METHOD  M_STATE_DORMANT
VAR_INPUT
END_VAR
Busy    := FALSE;
Done    := FALSE;
Aborted := FALSE;
Error   := FALSE;
FeedBack.InterventionRequest :=FALSE;
strStatus :='FB_UpperFeedInConveyor: No Error';
uiExecutingStep :=0;
uiResettingStep	:=0;
NoFirstBoxDiameter:= SecondBox:=FALSE;
tonUpperConveyorTimeOut.IN := FALSE;
tonUpperConveyorDelay.IN :=FALSE;
tonUpperTimeOut.IN :=FALSE;
tonUpperTimeOutFive.IN :=FALSE;
tonWaitSecondBoxArriveTimeout.IN :=FALSE;
TON_CheckHaveBox.IN :=false;
tonFeedAirBlowtime.IN :=false;
bSecondBoxInCameraPos := FALSE;
_bForceUpperCV_Use := false;
_Abort := _Executed := _Error:= _ResetCompleted:=_AbortCompleted:=FALSE;
iMoveConveyor := 0;
uiFirstBoxDiameterStep  :=0;
uiSecondBoxAirBlowStep	:=0;
_UniqueErrorCode :='0';
// 重置暫停相關變數
_bPaused := FALSE;
_bPauseEdge := FALSE;
IF Execute THEN
	RobotService_CheckUPCVServicedone := FALSE;
	eSTATE:=STATE_EXECUTING;
END_IF
END_METHOD

METHOD  M_STATE_ERROR
VAR_INPUT
END_VAR
ERROR :=TRUE;
Busy :=FALSE;
UniqueErrorCode:=_UniqueErrorCode;
SUPER^.Status := strStatus;
_fbDiameterMovement.Execute := FALSE;


Motor.List.UpCV.M_MotorStop(); 
OutPut.bCamara_Blow :=FALSE;

IF NOT Execute THEN	
eSTATE:=STATE_RESETTING;
END_IF
END_METHOD

METHOD  M_STATE_EXECUTING
VAR_INPUT
END_VAR

VAR_INST
	
	
END_VAR
VAR
	END_I: INT;
	
END_VAR
// 如果暫停中，直接返回不執行
IF _bPaused THEN
	RETURN;
END_IF

Busy :=TRUE;

//Conveyor motor control
CASE iMoveConveyor OF
	1:
	Motor.list.UpCV.M_MoveForward();
	Cylinder.List.fbUpCV_CamaraPress4.M_Retract(); //Feedin working , open the end to allow box feedin
	//OutPut.bCamara_Blow :=TRUE;
	-1:
	Motor.list.UpCV.M_MoveBackward();
	Cylinder.List.fbUpCV_CamaraPress4.M_Retract(); //Feedin working , open the end to allow box feedin
ELSE		
	Motor.list.UpCV.M_MotorStop();
	Cylinder.List.fbUpCV_CamaraPress4.M_Extend();// End feedin , block the conveyor in case no one push boxes in working area
	//OutPut.bCamara_Blow :=FALSE;		change use airflow to take photo before
END_CASE



CASE uiExecutingStep OF
	
0 : // StandBy
	TON_RecordTimer.IN := TRUE;
	iMoveConveyor:=0;
	tonUpperConveyorTimeOut.IN:=FALSE;
	tonUpperConveyorDelay.IN :=FALSE;
	tonUpperConveyorDelay.PT:=T#200MS;
	IF Info.NrOfBox=1 THEN
		SecondBox:=FALSE;
	ELSIF Info.NrOfBox=2 THEN
		SecondBox:=TRUE;	
	ELSE
	_Error := TRUE;
	  strStatus := 'FB_UpperFeedInConveyor Step 0: Data not correct';
	END_IF
	uiExecutingStep :=10;

10: //Prepare cylinders
	IF Cylinder.List.fbUpCV_FeedInPress1.xError THEN
		Cylinder.List.fbUpCV_FeedInPress1.M_Reset();
	END_IF
	IF Cylinder.List.fbUpCV_FeedInPress2.xError THEN
		Cylinder.List.fbUpCV_FeedInPress1.M_Reset();
	END_IF
	IF Cylinder.List.fbUpCV_DiameterPress.xError THEN
		Cylinder.List.fbUpCV_DiameterPress.M_Reset();
	END_IF
	IF Cylinder.List.fbUpCV_CamaraPress1.xError THEN
		Cylinder.List.fbUpCV_CamaraPress1.M_Reset();
	END_IF
	IF Cylinder.List.fbUpCV_CamaraPress2.xError THEN
		Cylinder.List.fbUpCV_CamaraPress2.M_Reset();
	END_IF
	IF Cylinder.List.fbUpCV_CamaraPress4.xError THEN
		Cylinder.List.fbUpCV_CamaraPress4.M_Reset();
	END_IF
	IF Cylinder.List.fbUpCV_Block1.xError THEN
		Cylinder.List.fbUpCV_Block1.M_Reset();
	END_IF
	IF Cylinder.List.fbUpCV_Block2.xError THEN
		Cylinder.List.fbUpCV_Block2.M_Reset();
	END_IF
	IF Cylinder.List.fbUpCV_Block3.xError THEN
		Cylinder.List.fbUpCV_Block3.M_Reset();
	END_IF
	IF Motor.List.UpCV.xError THEN
		Motor.List.UpCV.M_Reset();
	END_IF
	
	uiExecutingStep :=20;
	
20: //Prepare cylinders
	tonUpperTimeOut.IN :=TRUE;
	Cylinder.List.fbUpCV_FeedInPress1.M_Retract();		(* Cylinder.List.fbUpCV_FeedInPress1.M_Retract();*)	
	Cylinder.List.fbUpCV_FeedInPress2.M_Retract();		(*Cylinder.List.fbUpCV_FeedInPress2.M_Retract();*)
	Cylinder.List.fbUpCV_DiameterPress.M_Retract();		(*Cylinder.List.fbUpCV_DiameterPress.M_Retract();*)
	Cylinder.List.fbUpCV_CamaraPress1.M_Retract();		(*Cylinder.List.fbUpCV_CamaraPress1.M_Retract();*)		
	//Cylinder.List.fbUpCV_CamaraPress2.M_Retract();	(*Cylinder.List.fbUpCV_CamaraPress2.M_Retract();*)
	Cylinder.List.fbUpCV_CamaraPress4.M_Retract();		(*Cylinder.List.fbUpCV_CamaraPress4.M_Retract();*)	
	Cylinder.List.fbUpCV_Block1.M_Retract();			(*Cylinder.List.fbUpCV_Block1.M_Retract();*)
	Cylinder.List.fbUpCV_Block2.M_Retract();			(*Cylinder.List.fbUpCV_Block2.M_Retract();*)
	Cylinder.List.fbUpCV_Block3.M_Retract();			(*Cylinder.List.fbUpCV_Block3.M_Retract();*)

	//edit by Min 20250326
	IF Cylinder.List.fbUpCV_FeedInPress1.InRearPosition AND		
		Cylinder.List.fbUpCV_FeedInPress2.InRearPosition AND
		Cylinder.List.fbUpCV_DiameterPress.InRearPosition AND
		Cylinder.List.fbUpCV_CamaraPress1.InRearPosition AND
		Cylinder.List.fbUpCV_CamaraPress4.InRearPosition AND
		Cylinder.List.fbUpCV_Block1.InRearPosition AND
		Cylinder.List.fbUpCV_Block2.InRearPosition AND
		Cylinder.List.fbUpCV_Block3.InRearPosition THEN
		
		tonUpperTimeOut.IN :=FALSE;
		uiExecutingStep :=100;	
	END_IF
	IF tonUpperTimeOut.Q THEN
		_Abort :=TRUE;
		strStatus :='FB_UpperFeedInConveyor Step 20: Prepare Cylinder clear command timeout';
	END_IF
	
100:// Check No Box 
	IF Input.bUpCV_Block1Detect_Sensor OR 
	  Input.bUpCV_Block2Detect_Sensor OR
	  Input.bUpCV_BoxArrived_Sensor OR
	  Input.bUpCV_Block3Detect_Sensor THEN
	 	 IF NOT AddingBox THEN
		 _bForceUpperCV_Use := TRUE;		//force UpperCV for Backward CV use
	 	 uiExecutingStep :=110; //Try reverse conveyor 
			ELSE 
			  _Abort := TRUE;
		 	 strStatus := 'FB_UpperFeedInConveyor Step 100: Conveyor not ready , please remove boxes in front';
		  END_IF
	 ELSE
 		uiExecutingStep :=200; 
	 END_IF
110:
		iMoveConveyor:= -1;
		Cylinder.List.fbUpCV_CamaraPress2.M_Retract();
		tonReverseConveyorDelay.IN :=TRUE;
		uiExecutingStep :=120;

120:
		//tonFeedAirBlowtime.IN :=TRUE;
		IF tonReverseConveyorDelay.Q THEN
			iMoveConveyor :=0;
			uiExecutingStep :=130; 
		END_IF
130:
		tonReverseConveyorDelay.IN :=FALSE;
		IF Input.bUpCV_Block1Detect_Sensor OR 
		  Input.bUpCV_Block2Detect_Sensor OR
		  Input.bUpCV_BoxArrived_Sensor OR
	 	 Input.bUpCV_Block3Detect_Sensor THEN
			  _Abort := TRUE;
		 	 strStatus := 'FB_UpperFeedInConveyor Step 130: Conveyor not ready , please remove boxes in front';
		 ELSE
			uiExecutingStep :=140; 	 
		 END_IF		
140:
   		IF Motor.list.UpCV.InStopped THEN
			uiExecutingStep :=200;
		END_IF
200: // motor start and camera block up 
	_bForceUpperCV_Use := FALSE;		//release UpperCV force use 
	tonUpperConveyorTimeOut.IN:=TRUE;
	iMoveConveyor:=1;
	Cylinder.List.fbUpCV_CamaraPress2.M_Retract();
	Cylinder.List.fbUpCV_Block3.M_Extend();
	IF Cylinder.List.fbUpCV_Block3.InFrontPosition AND
		Cylinder.List.fbUpCV_CamaraPress2.InRearPosition THEN
		tonUpperConveyorTimeOut.IN:=FALSE;
		uiExecutingStep :=300;
	END_IF
	IF tonUpperConveyorTimeOut.Q THEN
	  _Error := TRUE;
	  strStatus := 'FB_UpperFeedInConveyor Step 200: Cylinder.List.fbUpCV_Block3 timeout';
	END_IF
		  
	  
300://Dtect camera sensor and wait first box arrive in camera position
	TON_CheckHaveBox.IN :=TRUE;
	tonUpperConveyorDelay.IN:=Input.bUpCV_Block3Detect_Sensor; //Delay a moment to make sure box move till end of block 	
	IF tonUpperConveyorDelay.Q THEN
			TON_CheckHaveBox.IN :=FALSE;
			Cylinder.List.fbUpCV_CamaraPress1.M_Extend(); //Press box 
			tonUpperConveyorDelay.IN := FALSE;
			uiExecutingStep :=400;			
	END_IF
	IF TON_CheckHaveBox.Q THEN	//if behind not have box feedback box = 0
		uiExecutingStep := 2700;
	END_IF
	
400:// Check pressing job done for first box in camera position	
	tonUpperTimeOut.IN :=TRUE;
	IF Cylinder.List.fbUpCV_CamaraPress1.InFrontPosition THEN
		tonUpperTimeOut.IN := FALSE;
		Cylinder.List.fbUpCV_CamaraPress2.M_Extend();
		uiExecutingStep :=450;		
	END_IF
	IF tonUpperTimeOut.Q THEN
		_Abort := TRUE;
		strStatus := 'FB_UpperFeedInConveyor Step 400: Cylinder.List.fbUpCV_CamaraPress1.M_MoveForward timeout';
	END_IF

450:// send first box camera signal
	
	tonFeedAirBlowtime.IN :=TRUE;
	OutPut.bCamara_Blow :=TRUE;
	IF tonFeedAirBlowtime.Q THEN
		tonFeedAirBlowtime.IN:=FALSE;
		OutPut.bCamara_Blow :=FALSE;
		FeedBack.FirstBoxCamera :=TRUE;
		TON_RecordFirstTimer.IN :=TRUE;
		uiExecutingStep :=460;
	END_IF
	

460: // Wait first box camera done
	// todo : timeout
	tonUpperTimeOutFive.IN :=TRUE;		//T#5S
	IF Info.FirstBoxCameraDone THEN
		tonUpperTimeOutFive.IN :=FALSE;
		//FeedBack.FirstBoxCamera :=FALSE;
		uiExecutingStep :=500;
	END_IF	
	IF tonUpperTimeOutFive.Q THEN
		_Abort :=TRUE;
		strStatus := 'FB_UpperFeedInConveyor Step 460: C# FirstBoxCameraDone timeout';
	END_IF
	
500://Let first box move forward
	TSaveFirstTime 	:= TON_RecordFirstTimer.ET;
	TON_RecordFirstTimer .IN :=FALSE;
	Cylinder.List.fbUpCV_CamaraPress1.M_Retract(); // release press
	Cylinder.List.fbUpCV_Block3.M_Retract();//release blocker todo : add description
	uiExecutingStep :=550;
	
550://check cylinder inrearposition		edit by Min 20250326
	tonUpperTimeOut.IN :=TRUE;
	IF Cylinder.List.fbUpCV_CamaraPress1.InRearPosition AND		
		Cylinder.List.fbUpCV_Block3.InRearPosition THEN
		
		uiExecutingStep :=600;
	END_IF
	IF tonUpperTimeOut.Q THEN
		_Abort := TRUE;
		strStatus := 'FB_UpperFeedInConveyor Step 550: Cylinder.List.fbUpCV_CamaraPress1 or Cylinder.List.fbUpCV_Block3 InRearPosition timeout';
	END_IF
	
600://Check if diameter camera needed
	tonUpperTimeOut.IN :=FALSE;
	tonUpperTimeOutFive.IN :=TRUE;
	IF Info.FirstBoxCameraDiameterRequest THEN
		tonUpperTimeOutFive.IN :=FALSE;
		uiExecutingStep :=700;
		ELSE
			IF SecondBox THEN
				tonUpperTimeOutFive.IN :=FALSE;
				NoFirstBoxDiameter:=TRUE;
				uiExecutingStep :=610;//Only if box 1 no need to measure diameter
			ELSE
				tonUpperTimeOutFive.IN :=FALSE;
				uiExecutingStep :=2400;	
			END_IF
	END_IF
	IF tonUpperTimeOutFive.Q THEN
		_Abort := TRUE;
		strStatus :='FB_UpperFeedInConveyor Step 600: C# FirstBoxCameraDiameterRequest timeout';
	END_IF
	
610: //Check Box 1 leave read code camera position
	tonUpperTimeOut.IN :=TRUE;
	tonUpperConveyorDelay.IN := NOT Input.bUpCV_Block3Detect_Sensor;
	IF tonUpperConveyorDelay.Q THEN
		tonUpperConveyorDelay.IN :=FALSE;
		uiExecutingStep :=620;
	END_IF
	IF tonUpperTimeOut.Q  THEN
		_Abort :=TRUE;
		strStatus :='FB_UpperFeedInConveyor Step 610: Input.bUpCV_Block3Detect_Sensor first box leave timeout';
	END_IF
	
620: // Leave Box 2				//timeout and Check InRearPositonEdit by Min 20250326	
		tonUpperTimeOut.IN :=FALSE;	
		IF SecondBox THEN			
			Cylinder.List.fbUpCV_CamaraPress2.M_Retract(); //Release press box
			Cylinder.List.fbUpCV_Block3.M_Extend(); //release blocker
			IF Cylinder.List.fbUpCV_CamaraPress2.InRearPosition AND Cylinder.List.fbUpCV_Block3.InFrontPosition THEN
				uiExecutingStep :=1100;
			END_IF
		END_IF
		
700: //Rise diameter blocker
	tonUpperTimeOut.IN :=TRUE;
	Cylinder.List.fbUpCV_Block2.M_Extend();
	IF Cylinder.List.fbUpCV_Block2.InFrontPosition THEN
		tonUpperTimeOut.IN :=FALSE;
		uiExecutingStep :=800;
	END_IF
	IF tonUpperTimeOut.Q THEN
		_Abort :=TRUE;
		strStatus :='FB_UpperFeedInConveyor Step 700: Cylinder.List.fbUpCV_Block2 MoveForward timeout';
	END_IF
800: // wait first box ready on diameter position
	tonUpperTimeOut.IN :=TRUE;
	tonUpperConveyorDelay.IN:=Input.bUpCV_Block2Detect_Sensor;
	IF tonUpperConveyorDelay.Q THEN
		tonUpperTimeOut.IN :=FALSE;
		tonUpperConveyorDelay.IN:=FALSE;
		Cylinder.List.fbUpCV_DiameterPress.M_Extend();
		
		IF SecondBox THEN	
			tonUpperTimeOut.IN :=FALSE;		
			Cylinder.List.fbUpCV_CamaraPress2.M_Retract();
			Cylinder.List.fbUpCV_Block3.M_Extend();
		END_IF
		uiExecutingStep :=1000;
	END_IF
	IF tonUpperTimeOut.Q THEN
		_Abort :=TRUE;
		strStatus :='FB_UpperFeedInConveyor Step 800: Box not at Input.bUpCV_Block2Detect_Sensor ';
	END_IF
	
1000: // Wait diameter blocker ready
	tonUpperTimeOut.IN :=TRUE;
	IF 	Cylinder.List.fbUpCV_DiameterPress.InFrontPosition THEN
		tonUpperTimeOut.IN :=FALSE;
		uiExecutingStep :=1100;
	END_IF
	IF tonUpperTimeOut.Q THEN
		_Abort :=TRUE;
		strStatus :='FB_UpperFeedInConveyor Step 1000: Cylinder.List.fbUpCV_DiameterPress MoveForward timeout';
	END_IF

1100: // Pick needle to diameter camera

		
		CASE uiFirstBoxDiameterStep OF
			
		0:
			IF NOT NoFirstBoxDiameter THEN
	  			_fbDiameterMovement.Execute := TRUE;
				uiFirstBoxDiameterStep:=100;
			ELSE
				uiFirstBoxDiameterStep:=9000;	
	  		END_IF
		
		100:
			IF _fbDiameterMovement.Busy THEN
				uiFirstBoxDiameterStep:=200;
			END_IF	
			
		200:
			tonUpperTimeOutFive.IN :=TRUE;
			 IF _fbDiameterMovement.PickDone THEN
				  tonUpperTimeOutFive.IN :=FALSE;
				  FeedBack.FirstBoxCameraDiameter:=TRUE;		  
			  END_IF
			 IF Info.FirstBoxCameraDiameterDone THEN
				tonUpperTimeOutFive.IN:=FALSE;
				 FeedBack.FirstBoxCameraDiameter:=FALSE;
			 	_fbDiameterMovement.bContinue:=TRUE;
			 	uiFirstBoxDiameterStep:=300;
			  END_IF
			 IF tonUpperTimeOutFive.Q THEN
				 _Error :=TRUE;
				 strStatus :='FB_UpperFeedInConveyor Step 1100: box1 diameter timeout';
			 END_IF
		300:
			 IF _fbDiameterMovement.Done THEN
				  uiFirstBoxDiameterStep:=9000;		  
			  END_IF	  
		
		9000:
				_fbDiameterMovement.bContinue:=FALSE;
				_fbDiameterMovement.Execute:=FALSE;
				Cylinder.List.fbUpCV_DiameterPress.M_Retract();
				Cylinder.List.fbUpCV_Block2.M_Retract();
				// first box leave	  
				
				IF bSecondBoxInCameraPos AND 
					Cylinder.List.fbUpCV_DiameterPress.InRearPosition AND
					Cylinder.List.fbUpCV_Block2.InRearPosition THEN
					
					uiExecutingStep :=1200;
				END_IF
		END_CASE
						
		
	  		IF SecondBox THEN
				tonWaitSecondBoxArriveTimeout.IN :=TRUE;
	  			tonUpperConveyorDelay.IN := Input.bUpCV_Block3Detect_Sensor;
 				IF tonUpperConveyorDelay.Q THEN								
					tonUpperConveyorDelay.IN:=FALSE;
					tonWaitSecondBoxArriveTimeout.IN :=FALSE;
					Cylinder.List.fbUpCV_CamaraPress2.M_Extend();
					Cylinder.List.fbUpCV_CamaraPress1.M_Extend();
//					bSecondBoxInCameraPos :=TRUE;
				END_IF	
	 		 ELSE
				 bSecondBoxInCameraPos:=TRUE;
	 		 END_IF
			 
		CASE uiSecondBoxAirBlowStep OF
			 0:
			 	IF 	Cylinder.List.fbUpCV_CamaraPress1.InFrontPosition AND 
					Cylinder.List.fbUpCV_CamaraPress2.InFrontPosition THEN
						uiSecondBoxAirBlowStep :=10;
				END_IF
			10:
				OutPut.bCamara_Blow :=TRUE;		//take photo need airflow before
				tonFeedAirBlowtime.IN :=TRUE;
					IF tonFeedAirBlowtime.Q THEN		
						tonFeedAirBlowtime.IN :=FALSE;
						OutPut.bCamara_Blow :=FALSE;
						FeedBack.SecondBoxCamera:=TRUE;
						TON_RecordSecondTimer.IN :=TRUE;
						uiSecondBoxAirBlowStep :=20;
					END_IF
			20:
				IF Info.SecondBoxCameraDone THEN
					uiSecondBoxAirBlowStep :=30;
					TSaveSecondTime := TON_RecordSecondTimer.ET;
				END_IF
			30:	
					
					
					TON_RecordSecondTimer.IN :=FALSE;
					bSecondBoxInCameraPos:=TRUE;	
			
		END_CASE
		
//			IF Cylinder.List.fbUpCV_CamaraPress1.InFrontPosition AND 
//				Cylinder.List.fbUpCV_CamaraPress2.InFrontPosition THEN
//				OutPut.bCamara_Blow :=TRUE;		//take photo need airflow before
//				tonFeedAirBlowtime.IN :=TRUE;
//					IF tonFeedAirBlowtime.Q THEN		
//						tonFeedAirBlowtime.IN :=FALSE;
//						OutPut.bCamara_Blow :=FALSE;
//						FeedBack.SecondBoxCamera:=TRUE;	
//							IF Info.SecondBoxCameraDone THEN
//								bSecondBoxInCameraPos:=TRUE;	
//							END_IF	
//					END_IF
//			END_IF
	  
	  IF tonUpperConveyorTimeOut.Q THEN
			_Error :=TRUE;
			strStatus:='FB_UpperFeedInConveyor Step 1100: First box diameter timeout';		
		  
	  END_IF
		IF tonWaitSecondBoxArriveTimeout.Q THEN
			IF Input.bUpCV_ReLoadDetect_Sensor THEN
				_Error :=TRUE;
				strStatus:='FB_UpperFeedInConveyor Step 1100: Second box feedin to read code camera pos timeout';		
			ELSE
				tonUpperConveyorTimeOut.IN :=FALSE;
				SecondBox :=FALSE;
			END_IF	 
		END_IF

1200: 	// If first box leave diameter sensor , let second box go
		tonUpperTimeOut.IN :=TRUE;
		tonUpperConveyorDelay.PT:=T#600MS;		
		tonUpperConveyorDelay.IN := NOT Input.bUpCV_Block2Detect_Sensor;
		
		IF tonUpperConveyorDelay.Q THEN
			tonUpperConveyorDelay.IN :=FALSE;
			tonUpperTimeOut.IN :=FALSE;
			IF SecondBox AND INfo.SecondBoxCameraDiameterRequest THEN
				tonUpperTimeOut.IN :=FALSE;
				Cylinder.List.fbUpCV_Block2.M_Extend();
				Cylinder.List.fbUpCV_CamaraPress1.M_Retract();
				Cylinder.List.fbUpCV_Block3.M_Retract();
				uiExecutingStep :=1700;
			ELSE
				tonUpperTimeOut.IN :=FALSE;
				Cylinder.List.fbUpCV_CamaraPress1.M_Retract();
				Cylinder.List.fbUpCV_Block3.M_Retract();
				uiExecutingStep :=2400;	
			END_IF

		END_IF
		IF tonUpperTimeOut.Q THEN
			_Abort :=TRUE;
			strStatus :='FB_UpperFeedInConveyor Step 1200: First box still at Input.bUpCV_Block2Detect_Sensor';
		END_IF

1700: //Second box diameter request
		tonUpperTimeOut.IN :=TRUE;
		tonUpperConveyorDelay.IN :=Input.bUpCV_Block2Detect_Sensor;
		IF tonUpperConveyorDelay.Q THEN
			tonUpperTimeOut.IN :=FALSE;
			tonUpperConveyorDelay.IN :=FALSE;
			Cylinder.List.fbUpCV_DiameterPress.M_Extend();
			uiExecutingStep :=1800;
		END_IF
		IF tonUpperTimeOut.Q THEN
			_Abort :=TRUE;
			strStatus :='FB_UpperFeedInConveyor Step 1700: Input.bUpCV_Block2Detect_Sensor not have box';
		END_IF
1800: //wait second box in diameter position
		tonUpperTimeOut.IN :=TRUE;
		IF Cylinder.List.fbUpCV_DiameterPress.InFrontPosition THEN
			tonUpperTimeOut.IN :=FALSE;
			uiExecutingStep :=1900;
		END_IF
		IF tonUpperTimeOut.Q THEN
			_Abort :=TRUE;
			strStatus :='FB_UpperFeedInConveyor Step 1800: Cylinder.List.fbUpCV_DiameterPress MoveForward timeout';
			
		END_IF
		
1900:
		tonUpperTimeOutFive.IN :=TRUE;
		_fbDiameterMovement.Execute :=TRUE	;	
		IF _fbDiameterMovement.PickDone THEN
			tonUpperTimeOutFive.IN :=FALSE;
			FeedBack.SecondBoxCameraDiameter:=TRUE;
			uiExecutingStep :=2000;
		END_IF
		IF tonUpperTimeOutFive.Q THEN
			_Abort :=TRUE;
			strStatus :='FB_UpperFeedInConveyor Step 1900: C# DiameterMovement Pickdone timeout';
		END_IF
2000:	//check Second Box CamaraDone
		tonUpperTimeOutFive.IN :=TRUE;
		IF info.SecondBoxCameraDiameterDone THEN
			tonUpperTimeOutFive.IN :=FALSE;
			FeedBack.SecondBoxCameraDiameter:=FALSE;
			_fbDiameterMovement.bContinue:=TRUE;
			uiExecutingStep :=2100;
		END_IF
		IF tonUpperTimeOutFive.Q THEN
			_Abort :=TRUE;
			strStatus :='FB_UpperFeedInConveyor Step 2000: C# SecondBoxCameraDiameterDone timeout';
		END_IF		
2100:	
		tonUpperTimeOutFive.IN :=TRUE;
		IF _fbDiameterMovement.Done THEN
			tonUpperTimeOutFive.IN :=FALSE;
			_fbDiameterMovement.Execute:=FALSE;
			uiExecutingStep :=2150;
		END_IF
		IF tonUpperTimeOutFive.Q THEN
			_Abort :=TRUE;
			strStatus :='FB_UpperFeedInConveyor Step 2100: _fbDiameterMovement Done timeout';
		END_IF
2150:
		IF  Input.bUpCV_BoxArrived_Sensor  AND 
			NOT Input.bUpCV_Block1Detect_Sensor  THEN
			uiExecutingStep :=2200;
		END_IF
2200:	// release box 2 from diameter camera pos
		tonUpperTimeOut.IN :=TRUE;
		tonUpperConveyorDelay.PT:=T#100MS;
		tonUpperConveyorDelay.IN := NOT Input.bUpCV_Block1Detect_Sensor ;
		IF tonUpperConveyorDelay.Q THEN	
			tonUpperConveyorDelay.IN := FALSE;
			Cylinder.List.fbUpCV_Block1.M_Extend();
			Cylinder.List.fbUpCV_DiameterPress.M_Retract();		
			Cylinder.List.fbUpCV_Block2.M_Retract();
			uiExecutingStep :=2300;
		END_IF
		IF tonUpperTimeOut.Q THEN
			_Error :=TRUE;
			strStatus := 'FB_UpperFeedInConveyor Step 2200: There is a box on Input.bUpCV_Block1Detect_Sensor ';
		END_IF
		
		
2300:
		tonUpperTimeOut.IN :=TRUE;
		IF 	Cylinder.List.fbUpCV_DiameterPress.InRearPosition AND
			Cylinder.List.fbUpCV_Block1.InFrontPosition AND
			Cylinder.List.fbUpCV_Block2.InRearPosition THEN
			tonUpperTimeOut.IN :=FALSE;
			uiExecutingStep :=2500;
		END_IF	
		IF tonUpperTimeOut.Q THEN
			_Error :=TRUE;
			strStatus :='FB_UpperFeedInConveyor Step 2300: BlockBox1 MoveForward or BlockBox2 MoveBackward or DiameterMeasurementPressBox MoveBackward timeout';
		END_IF
2400:	//Check Box1 in FeedInBox1Detecting and Box2 leave BlockBox2Detecting
		
		tonUpperConveyorDelay.PT:=T#100MS;
		tonUpperConveyorDelay.IN := Input.bUpCV_BoxArrived_Sensor ;
		
		IF  tonUpperConveyorDelay.Q AND NOT Input.bUpCV_Block1Detect_Sensor  THEN
			tonUpperConveyorDelay.IN:=FALSE;
			Cylinder.List.fbUpCV_CamaraPress1.M_Retract();
			Cylinder.List.fbUpCV_Block3.M_Retract();
			Cylinder.List.fbUpCV_Block1.M_Extend();
			uiExecutingStep :=2500;
		END_IF
		
2500:	// Check Box1 in FeedInBox1Sensor and Box2 in BlockBox1Sensor
		tonUpperTimeOutFive.IN :=TRUE;
		tonUpperConveyorDelay.PT:=T#300MS;
		tonUpperConveyorDelay.IN := Input.bUpCV_BoxArrived_Sensor  AND 
		(Input.bUpCV_Block1Detect_Sensor  OR NOT SecondBox);
		
		IF tonUpperConveyorDelay.Q THEN
			tonUpperTimeOutFive.IN :=FALSE;
			tonUpperConveyorDelay.IN :=FALSE;
			Cylinder.List.fbUpCV_FeedInPress1.M_Extend();
			IF SecondBox THEN
				Cylinder.List.fbUpCV_FeedInPress2.M_Extend();
			END_IF
			uiExecutingStep :=2600;
		END_IF
		IF tonUpperTimeOutFive.Q THEN
			_Error :=TRUE;
			strStatus :='FB_UpperFeedInConveyor Step 2500: FeedInBox1Detecting not have a box';
		END_IF
2600:
		tonUpperConveyorDelay.PT:=T#500MS;
		tonUpperTimeOut.IN := TRUE;
		tonUpperConveyorDelay.IN :=  Cylinder.List.fbUpCV_FeedInPress1.InFrontPosition AND
		 (Cylinder.List.fbUpCV_FeedInPress2.InFrontPosition OR NOT SecondBox);		
//		IF tonUpperConveyorDelay.IN THEN
//			iMoveConveyor:=0;
//			//Motor.list.UpCV.M_StopMotor();
//		END_IF
		IF tonUpperConveyorDelay.Q THEN
			iMoveConveyor:=0;
			tonUpperTimeOut.IN :=FALSE;
			tonUpperConveyorDelay.IN :=FALSE;
			 Cylinder.List.fbUpCV_FeedInPress1.M_Retract();
			IF SecondBox THEN
				Cylinder.List.fbUpCV_FeedInPress2.M_Retract();
			END_IF
			uiExecutingStep :=2700;
		END_IF	
		IF tonUpperTimeOut.Q THEN
			_Error :=TRUE;
			strStatus :='FB_UpperFeedInConveyor Step 2600: Cylinder.List.fbUpCV_FeedInPress1 or Cylinder.List.fbUpCV_FeedInPress2 MoveForward timeout';
		END_IF
2700:
		tonUpperTimeOut.IN :=TRUE;
		IF TON_CheckHaveBox.IN THEN	// conveyor behind not have box feedback 0
			FeedBack.ActualNrOfBox:=0;
		ELSIF SecondBox THEN
			FeedBack.ActualNrOfBox:=2;
			ELSE
			FeedBack.ActualNrOfBox:=1;	
		END_IF
		//Cylinder.List.fbUpCV_Block1.M_Retract();
		//Cylinder.List.fbUpCV_CamaraPress2.M_Retract();
		IF NOT input.bUpCV_ReLoadDetect_Sensor  THEN
			FeedBack.InterventionRequest :=TRUE;
		END_IF
		IF// Cylinder.List.fbUpCV_Block1.InRearPosition AND
			 Cylinder.List.fbUpCV_FeedInPress1.InRearPosition AND
			Cylinder.List.fbUpCV_FeedInPress2.InRearPosition THEN
			//Cylinder.List.fbUpCV_CamaraPress2.InRearPosition THEN
			tonUpperTimeOut.IN :=FALSE;
			uiExecutingStep := 2800;
		END_IF	
		IF tonUpperTimeOut.Q THEN 
			_Error :=TRUE;
			strStatus :='FB_UpperFeedInConveyor Step 2700: FeedInPressBox1Cylinder or FeedInPressBox2Cylinder or ReadCodePressBox2Cylinder MoveBackward timeout';
		END_IF
		
2800:	//TO check the camera photo speed recoeding time
	TSaveTime 		:= TON_RecordTimer.ET;
	tRecordTimer[iArrayNumber] 			:=TSaveTime;
	tRecordFirstTimer[iArrayNumber] 	:=TSaveFirstTime;
	tRecordSecondTimer[iArrayNumber] 	:=TSaveSecondTime;
	uiExecutingStep := 2900;
2900:
	iArrayNumber := iArrayNumber+1;
	TON_RecordTimer.IN := FALSE;
	IF iArrayNumber >= 101 THEN
		bResetRecordInfo 	:=TRUE;
		iArrayNumber 		:=1;
	END_IF
	uiExecutingStep := 9999;
9999:
	bResetRecordInfo :=FALSE;
	TON_CheckHaveBox.IN :=FALSE;
	_Executed := TRUE;
				
END_CASE
	
	
IF NOT Execute THEN
	eState:=STATE_RESETTING;
END_IF
IF _Error THEN
	//FUN_UniqueErrorCodeGenerator(iErrorID := ErrorID,UinqueErrorCode=>_UniqueErrorCode);
	eState:=STATE_ERROR;
END_IF
IF _Abort OR Abort THEN
	//FUN_UniqueErrorCodeGenerator(iErrorID := ErrorID,UinqueErrorCode=>_UniqueErrorCode);
	eSTATE:=STATE_ABORTING;
END_IF
IF _Executed THEN
	eSTATE:=STATE_Done;
END_IF
END_METHOD

METHOD  M_STATE_RESETTING
VAR_INPUT
END_VAR
Error :=_Error;
Done :=_Executed;

tonUpperTimeOut.IN:=TRUE;
Motor.List.UpCV.M_MotorStop();

IF tonUpperTimeOut.Q OR NOT _Error THEN
	CASE uiResettingStep OF
		0: 
			IF _Error THEN
				Cylinder.List.fbUpCV_Block1.M_Retract();
			END_IF
			Cylinder.List.fbUpCV_FeedInPress1 .M_Retract();	
			Cylinder.List.fbUpCV_FeedInPress2.M_Retract();
			Cylinder.List.fbUpCV_DiameterPress.M_Retract();
			Cylinder.List.fbUpCV_CamaraPress1.M_Retract();	
			//UpperReadCodePressBox2Cylinder.M_Retract();	
			Cylinder.List.fbUpCV_Block2.M_Retract();	
			Cylinder.List.fbUpCV_Block3.M_Retract();	
			Cylinder.List.fbUpCV_CamaraPress4.M_Retract();
			OutPut.bCamara_Blow :=FALSE;
			_fbDiameterMovement.Execute := FALSE;
			_fbDiameterMovement.bContinue:=FALSE;
			FeedBack.InterventionRequest :=FALSE;
			FeedBack.FirstBoxCamera :=FALSE;
			FeedBack.FirstBoxCameraDiameter :=FALSE;
			FeedBack.SecondBoxCamera :=FALSE;
			FeedBack.SecondBoxCameraDiameter :=FALSE;

		
			uiResettingStep:=9999;
		
		9999:
			_ResetCompleted:=TRUE;
	END_CASE
END_IF
IF _ResetCompleted THEN
	eSTATE:=STATE_DORMANT;
END_IF
END_METHOD

END_FUNCTION_BLOCK

// ---- Library/20_MachineUnits/21_StorageArea/Service/FB_AddBoxes_v2.TcPOU
FUNCTION_BLOCK FB_AddBoxes_v2 EXTENDS FB_ObjectBase_V2
VAR_INPUT
//	UpperBoxRefillDetection		:REFERENCE TO FB_Sensor;
//	RackPusherCylinder			:REFERENCE TO FB_Cylinder;
//	RackMotor					:REFERENCE TO FB_RackMotor_V2;
//	bUpperLayerFeedInConveyor	:REFERENCE TO FB_Motor;
	Cylinder 	: REFERENCE TO UNI_CylinderList;
	Motor	 	: REFERENCE TO UNI_MotorList;
	Input 	 	: REFERENCE TO ST_InputTable;
	OutPut	 	: REFERENCE TO ST_OutputTable;
	CurrentData      : ST_SetupPara;

	ERackState	:E_RackState;
	bClearInterventionRequest : BOOL;
	_bForceUpperCV_Use		:BOOL;
END_VAR
VAR_OUTPUT
	InterventionRequest	 : BOOL;
	FeedingBoxes		:BOOL;
END_VAR
VAR
	RackMotorStationTable   : ARRAY[0..9] OF st_StationPositions;
	uiMaxRackStation :INT :=10;
//	eState :E_MethodStatus_Basic;
//	uiExecutingStep : UDINT; // This var is used to been controll STATE_EXECUTING process.
//	uiResettingStep : UDINT;
//	uiAbortingStep : UDINT;
//	_Executed :BOOL; // Executing process completed.
//	_Error : BOOL; // FB has an error.
//	_ResetCompleted : BOOL; // FB resetting completed.
//	_AbortCompleted : BOOL; // FB aborting completed.	

	tonAddBoxTimeOut	:TON;
	tonDetectSensor		:TON;
	tonConveyorTimeOut	:TON;
	tonFeedInUseAddBoxesDelay :TON;
	strStatus	:STRING;
//	_Abort		:BOOL;
	CurrStation : UINT;
	bInterventionRequest	 : BOOL;
	trigClearInterventionRequest : R_TRIG;
	_bClearInterventionRequestLast :BOOL;
	ftrigRackStateLeaveFeedBox		:F_Trig;
	_UniqueErrorCode : STRING;
	_RetryCompleted	 : BOOL; // FB Aboted STATE use

	// ===== Pause / Resume framework =====
	_bPaused					: BOOL;
	_bPauseEdge					: BOOL;

	// 計時器活動狀態保存
	bWasActive_tonAddBoxTimeOut			: BOOL;
	bWasActive_tonDetectSensor			: BOOL;
	bWasActive_tonConveyorTimeOut		: BOOL;
	bWasActive_tonFeedInUseAddBoxesDelay : BOOL;

	// 計時器剩餘時間保存
	tRemaining_tonAddBoxTimeOut			: TIME;
	tRemaining_tonDetectSensor			: TIME;
	tRemaining_tonConveyorTimeOut		: TIME;
	tRemaining_tonFeedInUseAddBoxesDelay : TIME;

	// 恢復後使用調整 PT 旗標 (Q 觸發或被外部關掉就清除)
	bUseAdjustedPT_tonAddBoxTimeOut		: BOOL;
	bUseAdjustedPT_tonDetectSensor		: BOOL;
	bUseAdjustedPT_tonConveyorTimeOut	: BOOL;
	bUseAdjustedPT_tonFeedInUseAddBoxesDelay : BOOL;

	// 馬達/輸出狀態保存
	bSaved_MoveConveyor			: BOOL;

	// 從 EXECUTING.VAR_INST 提到 FB-level (A01_PauseControl 需 access)
	bMoveConveyor				: BOOL;
END_VAR

A00_BasicUnits();
A01_PauseControl();

// 暫停時不執行狀態機
IF NOT _bPaused THEN
	SUPER^.A10_StateControl();
END_IF

ACTION A00_BasicUnits:
// 計時器 PT 設定 - 恢復後使用剩餘時間,完成後切回原 PT
IF bUseAdjustedPT_tonAddBoxTimeOut THEN
	tonAddBoxTimeOut(PT := tRemaining_tonAddBoxTimeOut);
	IF tonAddBoxTimeOut.Q OR NOT tonAddBoxTimeOut.IN THEN
		bUseAdjustedPT_tonAddBoxTimeOut := FALSE;
	END_IF
ELSE
	tonAddBoxTimeOut(PT:=T#120S);
END_IF

IF bUseAdjustedPT_tonDetectSensor THEN
	tonDetectSensor(PT := tRemaining_tonDetectSensor);
	IF tonDetectSensor.Q OR NOT tonDetectSensor.IN THEN
		bUseAdjustedPT_tonDetectSensor := FALSE;
	END_IF
ELSE
	tonDetectSensor(PT:=T#1S);
END_IF

IF bUseAdjustedPT_tonConveyorTimeOut THEN
	tonConveyorTimeOut(PT := tRemaining_tonConveyorTimeOut);
	IF tonConveyorTimeOut.Q OR NOT tonConveyorTimeOut.IN THEN
		bUseAdjustedPT_tonConveyorTimeOut := FALSE;
	END_IF
ELSE
	tonConveyorTimeOut(PT:=T#5S);
END_IF

IF bUseAdjustedPT_tonFeedInUseAddBoxesDelay THEN
	tonFeedInUseAddBoxesDelay(PT := tRemaining_tonFeedInUseAddBoxesDelay);
	IF tonFeedInUseAddBoxesDelay.Q OR NOT tonFeedInUseAddBoxesDelay.IN THEN
		bUseAdjustedPT_tonFeedInUseAddBoxesDelay := FALSE;
	END_IF
ELSE
	tonFeedInUseAddBoxesDelay(PT:=T#1S);
END_IF

ErrorID := 2700;

InterventionRequest:=bInterventionRequest;
ftrigRackStateLeaveFeedBox(CLK := (eRackState = E_RackState.FeedBox));
IF ftrigRackStateLeaveFeedBox.Q THEN
	bInterventionRequest:=FALSE;
END_IF

FeedingBoxes := eRackState=E_RackState.FeedBox;
END_ACTION

ACTION A01_PauseControl:
// A01_PauseControl - 暫停控制邏輯
// 依 PauseResume_Implementation_Guide.md 標準框架實作
// 控制對象: tonAddBoxTimeOut/tonDetectSensor/tonConveyorTimeOut/tonFeedInUseAddBoxesDelay 4 個計時器
//          Motor.List.UpCV (DC 馬達, 透過 bMoveConveyor 控制)
//          arAxisCtrl_gb[AxisNo.RackMotor] (伺服軸)

Paused := _bPaused;

// 只在執行狀態處理暫停
IF eState <> STATE_EXECUTING THEN
	_bPaused := FALSE;
	_bPauseEdge := FALSE;
	RETURN;
END_IF

// ===== 進入暫停 (上升邊緣) =====
IF Pause AND NOT _bPauseEdge THEN
	_bPauseEdge := TRUE;

	IF NOT _bPaused THEN
		_bPaused := TRUE;

		// 保存計時器活動狀態和剩餘時間
		bWasActive_tonAddBoxTimeOut := tonAddBoxTimeOut.IN;
		tRemaining_tonAddBoxTimeOut := T#120S - tonAddBoxTimeOut.ET;

		bWasActive_tonDetectSensor := tonDetectSensor.IN;
		tRemaining_tonDetectSensor := T#1S - tonDetectSensor.ET;

		bWasActive_tonConveyorTimeOut := tonConveyorTimeOut.IN;
		tRemaining_tonConveyorTimeOut := T#5S - tonConveyorTimeOut.ET;

		bWasActive_tonFeedInUseAddBoxesDelay := tonFeedInUseAddBoxesDelay.IN;
		tRemaining_tonFeedInUseAddBoxesDelay := T#1S - tonFeedInUseAddBoxesDelay.ET;

		// 停止所有計時器 (避免暫停期間 Timeout)
		tonAddBoxTimeOut.IN := FALSE;
		tonDetectSensor.IN := FALSE;
		tonConveyorTimeOut.IN := FALSE;
		tonFeedInUseAddBoxesDelay.IN := FALSE;

		// 保存上層輸送帶狀態
		bSaved_MoveConveyor := bMoveConveyor;

		// 停止上層輸送帶 (DC 馬達)
		Motor.List.UpCV.M_MotorStop();

		// 注意:RackMotor 不主動 halt
		// (1) 本 codebase 軸 API 沒有 Admin.Stop,要 halt 必須切 _OpMode.en := ModeAH 但 resume 後要重 issue 太複雜
		// (2) 暫停期間 SUPER^.A10_StateControl 不執行,軸完成 in-flight 移動後 state machine 不會推進
		// (3) Resume 時 step 210/610 直接看到 CmdDone 立即過 step,行為等價
	END_IF
END_IF

// ===== 離開暫停 (下降邊緣) - 必須等 Start 按鈕觸發 =====
IF NOT Pause AND _bPauseEdge AND GVL_ADS.OpPannel_Status.StartBtnStatus THEN
	_bPauseEdge := FALSE;

	IF _bPaused THEN
		_bPaused := FALSE;

		// 恢復上層輸送帶: 透過 bMoveConveyor 在 EXECUTING preamble 自動 M_MoveForward
		bMoveConveyor := bSaved_MoveConveyor;

		// 軸:暫停時沒主動 halt,resume 不需要 restore (對應上方 pause 注意事項)

		// 恢復計時器 (使用剩餘時間,A00 完成後切回原 PT)
		IF bWasActive_tonAddBoxTimeOut THEN
			bUseAdjustedPT_tonAddBoxTimeOut := TRUE;
			tonAddBoxTimeOut.IN := TRUE;
		END_IF

		IF bWasActive_tonDetectSensor THEN
			bUseAdjustedPT_tonDetectSensor := TRUE;
			tonDetectSensor.IN := TRUE;
		END_IF

		IF bWasActive_tonConveyorTimeOut THEN
			bUseAdjustedPT_tonConveyorTimeOut := TRUE;
			tonConveyorTimeOut.IN := TRUE;
		END_IF

		IF bWasActive_tonFeedInUseAddBoxesDelay THEN
			bUseAdjustedPT_tonFeedInUseAddBoxesDelay := TRUE;
			tonFeedInUseAddBoxesDelay.IN := TRUE;
		END_IF
	END_IF
END_IF

// 邊緣重置
IF NOT Pause THEN
	_bPauseEdge := FALSE;
END_IF
END_ACTION

METHOD PRIVATE M_CheckCommand : BOOL
VAR_INPUT
END_VAR
M_CheckCommand	:= true;
END_METHOD

METHOD PRIVATE M_GetCurrentStation : BOOL
VAR
	i : UINT;
	SetPos	 :LREAL;
END_VAR

VAR_OUTPUT
	uiCurrentStation	:UINT;
END_VAR
//SetPos := THIS^.fbMotor.NcToPlc.SetPos;
SetPos := arAxisCtrl_gb[AxisNo.RackMotor].Admin.Axis.NcToPlc.SetPos;
M_RefreshStationPos();
//IF  THIS^.fbMotor.Status.Homed THEN
IF arAxisCtrl_gb[AxisNo.RackMotor].Admin.Axis.Status.Homed THEN
	FOR i:=0 TO 9 BY 1 DO 
		IF SetPos> RackMotorStationTable[i].Position-5 AND SetPos< RackMotorStationTable[i].Position+5 THEN // Range should be confirm
			uiCurrentStation :=i;
			M_GetCurrentStation :=TRUE;
			RETURN;
		END_IF
	END_FOR
	
	uiCurrentStation:=99;
	M_GetCurrentStation :=FALSE;
ELSE
	M_GetCurrentStation :=FALSE;
	uiCurrentStation:=99;
END_IF
END_METHOD

METHOD PRIVATE M_MoveToStation : BOOL
VAR_INPUT
	uiStation : UINT;
END_VAR
VAR
	bDone	:BOOL;
	uiTargetPosition	:LREAL ;
END_VAR
M_RefreshStationPos();
IF uiStation>=0 AND uiStation <10 THEN
	uiTargetPosition :=RackMotorStationTable[uiStation].Position;
	
	arAxisCtrl_gb[AxisNo.RackMotor].PosMode.Acc := CurrentData.Axes.RackMotor.HalfAuto.Acceleration;
	arAxisCtrl_gb[AxisNo.RackMotor].PosMode.Dec := CurrentData.Axes.RackMotor.HalfAuto.Deceleration;
	arAxisCtrl_gb[AxisNo.RackMotor].PosMode.Jerk := CurrentData.Axes.RackMotor.HalfAuto.Jerk;
	arAxisCtrl_gb[AxisNo.RackMotor].PosMode.Velocity := CurrentData.Axes.RackMotor.HalfAuto.Velocity;
	arAxisCtrl_gb[AxisNo.RackMotor].PosMode.Position := uiTargetPosition;
	
//	THIS^.fbMotor.MoveAbs(lrPosition	:=uiTargetPosition,
//						lrVelocity 		:=GVL.MotorCore[AxisNo.RackMotor].VCC,
//						lrAcceleration	:=GVL.MotorCore[AxisNo.RackMotor].ACC,
//						lrDeceleration	:=GVL.MotorCore[AxisNo.RackMotor].DCC,
//						lrJerk			:=GVL.MotorCore[AxisNo.RackMotor].Jerk,
//						BufferMode		:=MC_BufferMode.MC_Aborting);
	//THIS^.fbMotor.GetCmdDoneStatus(bMotionCmdDone=>bDone);
ELSE
	M_MoveToStation :=FALSE;
	RETURN;
END_IF
END_METHOD

METHOD PRIVATE M_RefreshStationPos : BOOL
VAR_INPUT
END_VAR
VAR
	i: UINT;
	position : ST_PositionTable;
END_VAR
FOR i := 0 TO 9 DO
	position :=FUN_GetPositionTableData(PositionName:='W',Index:=i,Clip:=0);
RackMotorStationTable[i].Position:= position.X_Pos;
END_FOR
	M_RefreshStationPos :=TRUE;

// todo : update position of each stations
//FOR i:=1 TO 200 BY 1 DO
//	FOR iIndex:=0 TO 9 BY 1 DO
//		IF 		
//			DAS_CoreSys.MachineControl.CurrentData.PositionTable[i].Index= iIndex AND
//			DAS_CoreSys.MachineControl.CurrentData.PositionTable[i].Zone ='W' THEN
//			RackMotorStationTable[iIndex].Position := DAS_CoreSys.MachineControl.CurrentData.PositionTable[i].X_Pos;

//			StationsPosition[iIndex]:=RackMotorStationTable[i].Position;
//		ELSE
//			M_RefreshStationPos :=FALSE;
//		END_IF
//	END_FOR
//END_FOR
END_METHOD

METHOD  M_STATE_ABORTED
VAR_INPUT
END_VAR
Error :=TRUE;
Busy :=FALSE;
Done := FALSE;
Status :=strStatus;
UniqueErrorCode:=_UniqueErrorCode;
uiAbortingStep := 0;
_AbortCompleted := FALSE;


CASE uiExecutingStep OF
	0, 10:
			// init 階段 abort -> 從頭重跑
			_RetryCompleted := TRUE;
			uiExecutingStep := 0;
			strStatus := 'FB_AddBoxes_v2 init step: retrying from 0';

	100:
			_RetryCompleted := TRUE;
			uiExecutingStep := 100;
			strStatus := 'FB_AddBoxes_v2 Step 100: no error , retrying';

	200, 210:
			// 軸移動階段 abort -> 退到 200 重新發送移動指令
			_RetryCompleted := TRUE;
			uiExecutingStep := 200;
			strStatus := 'FB_AddBoxes_v2 Step 200/210: no error , retrying motion';

	300:
			_RetryCompleted := TRUE;
			uiExecutingStep := 300;
			strStatus := 'FB_AddBoxes_v2 Step 300: no error , retrying';

	400, 500:
			// sensor 檢查階段 abort -> 退到 400 重新檢查
			_RetryCompleted := TRUE;
			uiExecutingStep := 400;
			strStatus := 'FB_AddBoxes_v2 Step 400/500: no error , retrying refill check';

	600, 610:
			// 歸零移動階段 abort -> 退到 600 重新發送
			_RetryCompleted := TRUE;
			uiExecutingStep := 600;
			strStatus := 'FB_AddBoxes_v2 Step 600/610: no error , retrying home move';

	1000, 1100:
			// 收尾階段 abort -> 從 1000 完成停輸送帶
			_RetryCompleted := TRUE;
			uiExecutingStep := 1000;
			strStatus := 'FB_AddBoxes_v2 Step 1000/1100: no error , finishing';
ELSE
			// 未涵蓋的 step -> 不允許續作,只能放開 Execute 走 RESETTING 重跑
			_RetryCompleted := FALSE;
			strStatus := 'FB_AddBoxes_v2 unexpected step at aborted';
END_CASE

IF NOT Execute THEN
	eState := STATE_RESETTING;
END_IF

IF Execute AND Reset AND _RetryCompleted THEN
	_Abort := Error := _Error := FALSE;
	eState:=STATE_EXECUTING;
END_IF
END_METHOD

METHOD  M_STATE_ABORTING
VAR_INPUT
END_VAR
CASE uiAbortingStep of
	 0:		// 清空參數
			tonAddBoxTimeOut.IN			 := FALSE;
			tonDetectSensor.IN			 := FALSE;
			tonConveyorTimeOut.IN		 := FALSE;
			tonFeedInUseAddBoxesDelay.IN := FALSE;
			_RetryCompleted := FALSE;
			Motor.List.UpCV.M_MotorStop();
			
			uiAbortingStep := 100;
			
	100:	// 確認軸、氣缸是否有報錯
			IF  NOT arAxisCtrl_gb[AxisNo.RackMotor].Admin.Axis.Status.Error AND 
				NOT Cylinder.List.fbStackPush.xError THEN
				uiAbortingStep := 200;	
			ELSIF arAxisCtrl_gb[AxisNo.RackMotor].Admin.Axis.Status.Error THEN
				arAxisCtrl_gb[AxisNo.RackMotor].Admin.ClearError := TRUE;
			ELSIF Cylinder.List.fbStackPush.xError THEN
				Cylinder.List.fbStackPush.M_Reset();
			END_IF
			IF arAxisCtrl_gb[AxisNo.RackMotor].Admin.ClearError THEN 
				arAxisCtrl_gb[AxisNo.RackMotor].Admin.ClearError := FALSE;
			END_IF
			
	200:	// 推盒氣缸往後，料架軸
			Cylinder.List.fbStackPush.M_Retract();
			arAxisCtrl_gb[AxisNo.RackMotor].Admin._OpMode.en := E_AXIS_MODE.ModeAH;
			uiAbortingStep:=9999;
		
	9999:	
			_AbortCompleted:=TRUE;
END_CASE

IF	 _AbortCompleted THEN
	eSTATE:=STATE_ABORTED;
END_IF
END_METHOD

METHOD  M_STATE_DONE
VAR_INPUT
END_VAR
Busy := FALSE;
Done := TRUE;
IF NOT Execute THEN
	eState := STATE_RESETTING;
END_IF
END_METHOD

METHOD  M_STATE_DORMANT
VAR_INPUT
END_VAR
VAR
END_VAR
Busy    := FALSE;
Done    := FALSE;
Aborted := FALSE;
Error   := FALSE;
strStatus  := 'No error';
uiExecutingStep := 0;
uiResettingStep := 0;
uiAbortingStep:=0;
_ResetCompleted := FALSE;
_RetryCompleted := FALSE;
_AbortCompleted := FALSE;
_Abort := _Executed := _Error:= _ResetCompleted:=_AbortCompleted:=FALSE;
tonAddBoxTimeOut.IN :=FALSE;
tonDetectSensor.IN:=FALSE;
tonFeedInUseAddBoxesDelay.IN :=FALSE;
_UniqueErrorCode :='0';

// 重置暫停相關變數
_bPaused := FALSE;
_bPauseEdge := FALSE;

IF Execute  THEN
	IF eRackState = E_RackState.FeedBox THEN
		eState:= STATE_ERROR;
		strStatus :='FB_AddBoxes_v2: Rack occupied by user Push FeedButton';
		
	ELSIF  Input.bUpCV_ReLoadDetect_Sensor THEN
		_Executed :=TRUE;
		eState	:= STATE_Done;
	ELSE
		eState := STATE_EXECUTING;
	END_IF	
END_IF
END_METHOD

METHOD  M_STATE_ERROR
VAR_INPUT
END_VAR
Error := TRUE;
Busy :=FALSE;
Status :=strStatus;
UniqueErrorCode:=_UniqueErrorCode;

IF NOT Execute THEN
	eSTATE :=STATE_RESETTING;
END_IF

// 對稱 ABORTED 的 retry: 維持 Execute + 按 Reset 從 step 0 重跑
// 目前唯一 ERROR 觸發點 (step 0 wrong command) 由此處重試
IF Execute AND Reset THEN
	_Error := FALSE;
	Error := FALSE;
	uiExecutingStep := 0;
	eSTATE := STATE_EXECUTING;
END_IF
END_METHOD

METHOD  M_STATE_EXECUTING
VAR_INPUT
END_VAR
VAR_INST
	uiTargetStation	: UINT;
END_VAR
VAR
	bMotionDone : BOOL;
	
END_VAR
// 暫停中直接返回
IF _bPaused THEN
	RETURN;
END_IF

Busy := TRUE;
IF NOT _bForceUpperCV_Use THEN
	IF bMoveConveyor THEN
		Motor.List.UpCV.M_MoveForward();
//	ELSE
//		Motor.List.UpCV.M_MotorStop();
	END_IF
END_IF
CASE uiExecutingStep OF			
	
	0:	//check command
		tonAddBoxTimeOut.IN:=FALSE;
		tonFeedInUseAddBoxesDelay.IN :=TRUE;
		
		IF M_CheckCommand() THEN
			IF tonFeedInUseAddBoxesDelay.Q THEN
				tonFeedInUseAddBoxesDelay.IN :=FALSE;
				uiExecutingStep	:= 10 ;
			END_IF
		ELSE
			strStatus := 'FB_AddBoxes_v2 Step 0: Wrong command, check the command setting';
			_Error := TRUE;
		END_IF
	10:
		IF 	NOT	Motor.List.UpCV.InBackWard THEN
			uiExecutingStep	:= 100 ;
		END_IF
		//todo : Add timeout
		
 	100:	//release cylinder, check rackmotor currentStation
		tonAddBoxTimeOut.IN:=TRUE;
		tonDetectSensor.IN:=FALSE;
		Cylinder.List.fbStackPush.M_Retract();
		M_GetCurrentStation(uiCurrentStation =>CurrStation);
		
		IF	Cylinder.List.fbStackPush.InRearPosition THEN
			 CASE CurrStation OF
				0 ,99 :
					uiTargetStation:=1;				
				1,2,3,4,5,6,7,8,9 :
					uiTargetStation :=CurrStation;	
				ELSE // Error
					strStatus := 'FB_AddBoxes_v2 Step 100: Station get Error';
                    _Abort := TRUE;
			 END_CASE
			 
			 IF NOT _Abort THEN
                tonAddBoxTimeOut.IN := FALSE;
                uiExecutingStep := 200;
             END_IF
		END_IF
		
		IF tonAddBoxTimeOut.Q THEN
			strStatus := 'FB_AddBoxes_v2 Step 100: RackPusher move back timeout';
            _Abort := TRUE;
		END_IF
		
	200:	//check rackmotor station 
		tonDetectSensor.IN :=FALSE;
		IF uiTargetStation<10 THEN
			M_MoveToStation(uiTargetStation);
			uiExecutingStep := 210;	
		ELSE
			uiExecutingStep := 500;	
		END_IF
		
	
	210:
		tonAddBoxTimeOut.IN:=TRUE;
		bMotionDone:= arAxisStatus_gb[AxisNo.RackMotor].Admin._OpModeAck = ModePosAbs AND arAxisStatus_gb[AxisNo.RackMotor].Admin.CmdDone;
	//	RackMotor.fbMotor.GetCmdDoneStatus(bMotionCmdDone=>bMotionDone);
		M_GetCurrentStation(uiCurrentStation =>CurrStation);
	//CurrStation:= RackMotor.P_CurrentStattion;
		IF bMotionDone AND uiTargetStation = CurrStation THEN
			tonAddBoxTimeOut.IN:=FALSE;
			uiExecutingStep := 300;	
		END_IF
		IF tonAddBoxTimeOut.Q THEN
			strStatus := 'FB_AddBoxes_v2 Step 210: Rackmotor moving timeout';
            _Abort := TRUE;
		END_IF
		
	300:	//Cylinder moveforward
		tonAddBoxTimeOut.IN:=TRUE;
		Cylinder.List.fbStackPush.M_Extend();
		//bUpperLayerFeedInConveyor.M_ForwardMotor('');
		bMoveConveyor :=TRUE; //Move conveyor motor forward
		IF  Motor.List.UpCV.InForWard THEN	// make sure upperCV release force use
			IF Cylinder.List.fbStackPush.InFrontPosition THEN
				tonAddBoxTimeOut.IN:=FALSE;
				uiExecutingStep := 400;
			END_IF
		END_IF
		IF tonAddBoxTimeOut.Q THEN
			strStatus := 'FB_AddBoxes_v2 Step 300: RackPusher move forward timeout';
            _Abort := TRUE;
		END_IF
		
	400:	//check refillsensor have refill
		tonDetectSensor.IN:= NOT Input.bUpCV_ReLoadDetect_Sensor;
		Cylinder.List.fbStackPush.M_Retract();
		IF Cylinder.List.fbStackPush.InRearPosition THEN
			IF Input.bUpCV_ReLoadDetect_Sensor THEN
				uiExecutingStep :=500;
			ELSIF tonDetectSensor.Q THEN
				uiTargetStation := CurrStation+1;		
				uiExecutingStep :=200;
			END_IF
		END_IF
		
	500:	//確認氣缸是否在後，Done
		tonAddBoxTimeOut.IN:=TRUE;
			//bUpperLayerFeedInConveyor.M_StopMotor(''); 
			//bMoveConveyor :=FALSE;// Stop Conveyor
			tonAddBoxTimeOut.IN:=FALSE;
			IF uiTargetStation>=9 THEN
				uiExecutingStep :=600;
			ELSE
				bMoveConveyor :=FALSE;
				Motor.List.UpCV.M_MotorStop();	
				uiExecutingStep :=1000;
			END_IF
		
		
		IF tonAddBoxTimeOut.Q THEN
			strStatus := 'FB_AddBoxes_v2 Step 500: RackPusher move back timeout';
            _Abort := TRUE;
		END_IF
	600:
		tonAddBoxTimeOut.IN:=FALSE	;
		 M_MoveToStation(0);
		 uiExecutingStep:=610;
		 
	610:	
		M_GetCurrentStation(uiCurrentStation =>CurrStation);
		tonAddBoxTimeOut.IN:=TRUE;
		bMotionDone:=arAxisStatus_gb[AxisNo.RackMotor].Admin._OpModeAck = ModePosAbs AND arAxisStatus_gb[AxisNo.RackMotor].Admin.CmdDone;
		IF bMotionDone AND 0 = CurrStation THEN
			bInterventionRequest	 :=TRUE;
			tonAddBoxTimeOut.IN:=FALSE	;
			bMoveConveyor :=FALSE;
			Motor.List.UpCV.M_MotorStop();	
			uiExecutingStep:=1000;
		END_IF
 		IF tonAddBoxTimeOut.Q THEN
			strStatus := 'FB_AddBoxes_v2 Step 610: RackPusher move back timeout';
            _Abort := TRUE;
		END_IF
	1000:
		bMoveConveyor :=FALSE;// Stop Conveyor
		uiExecutingStep:=1100;
		
	1100:		
		_Executed := TRUE;
	
		
//		strStatus := 'Rack is empty';
//		_Error :=TRUE;
	
	
END_CASE

IF NOT Execute THEN
	eSTATE :=STATE_RESETTING;
END_IF
IF _Executed THEN
	eSTATE := STATE_DONE;
END_IF
IF _Error THEN
	//FUN_UniqueErrorCodeGenerator(iErrorID := ErrorID,UinqueErrorCode=>_UniqueErrorCode);
	eSTATE:=STATE_ERROR;
END_IF
IF _Abort OR Abort THEN
	//FUN_UniqueErrorCodeGenerator(iErrorID := ErrorID,UinqueErrorCode=>_UniqueErrorCode);
	eSTATE:=STATE_ABORTING;
END_IF
END_METHOD

METHOD  M_STATE_RESETTING
VAR_INPUT
END_VAR

VAR
	bMotionDone : BOOL;
END_VAR
CASE uiResettingStep OF
	0:
		tonAddBoxTimeOut.IN:=FALSE;		
		tonDetectSensor.IN:=FALSE;
		Cylinder.List.fbStackPush.M_Retract();

		IF Cylinder.List.fbStackPush.InRearPosition THEN
		uiResettingStep :=100;
		END_IF
		
	100:
		arAxisCtrl_gb[AxisNo.RackMotor].Admin._OpMode.en := E_AXIS_MODE.ModeAH;
		//RackMotor.fbMotor.Stop(0,0);
		//RackMotor.fbMotor.GetCmdDoneStatus(bMotionCmdDone=>bMotionDone);
		Motor.List.UpCV.M_MotorStop();
		uiResettingStep := 200;

		
	200:
		 Error :=false;
		_ResetCompleted := TRUE;
END_CASE

IF _ResetCompleted THEN
	eState := STATE_DORMANT;
END_IF
END_METHOD

END_FUNCTION_BLOCK

// ---- Library/20_MachineUnits/21_StorageArea/Service/FB_BoxSupplyCtrl_v1.TcPOU
FUNCTION_BLOCK FB_BoxSupplyCtrl_v1 EXTENDS FB_ObjectBase_V2
VAR_INPUT
//    Execute    :BOOL;   // True : This prog will start.
//    Abort      :BOOL;   // True : This prog will be abort.
//    Reset      :BOOL;   // True : This prog will be reset.
//    ObjectName :STRING; // Set this fb name(About it's action)

//	SupplyBTN 				:REFERENCE TO FB_Button;			//2nd machine
//	RackMotor				:REFERENCE TO FB_RackMotor_V2;
//	BoxesPusherCylinder		:REFERENCE TO FB_Cylinder;


	Cylinder				:REFERENCE TO UNI_CylinderList;
	Motor					:REFERENCE TO UNI_MotorList;
	Input 					:REFERENCE TO ST_InputTable;
	Output					:REFERENCE TO ST_OutputTable;
	fbstorageHome			: REFERENCE TO FB_StorageHoming;
	StroageRegionMode 		:E_UnitMode;
	bAddsBoxRequest 		: BOOL;
	AddBoxes_Status			:ST_AutoAddsBoxesStatus;
	AddBoxes_Ctrl			:ST_AutoAddsBoxesCommand;
	CurrentData 			: ST_SetupPara;
	
END_VAR

VAR_OUTPUT
	RackState : E_RackState;
	AxisRackMotorBTNHomeRequest	:BOOL;
//    Busy    :BOOL;        // True : This prog is running.
//    Done    :BOOL;        // True : Command has been executed.
//    Aborted :BOOL;        // True : This prog is aborted.
//    Error   :BOOL;        // True : This prog has an error.
//    ErrorID :UINT;       // Output ErrorID
//    Status  :T_MaxString; // Output this prog status by string(255bytes)
END_VAR

VAR
//    eState :E_MethodStatus_Basic;
//	uiExecutingStep : UDINT; // This var is used to been controll STATE_EXECUTING process.
//	uiResettingStep : UDINT;
//	uiAbortingStep : UDINT;
//	_Executed :BOOL; // Executing process completed.
//	_Error : BOOL; // FB has an error.
//	_ResetCompleted : BOOL; // FB resetting completed.
//	_AbortCompleted : BOOL; // FB aborting completed.
	RackMotorStationTable   : ARRAY[0..9] OF st_StationPositions;
	uiMaxRackStation :INT :=10;
//	_Abort		: BOOL;
	strStatus	: STRING;
	uiResumeStep : UINT;
	ExcutingStep :E_RackState;
	ftrigBTN		:F_TRIG;			// 放開瞬間判讀短按
	tonLongPress	:TON;				// 長按 3s 啟動 NG 軌道後退
	bLongPressActive	:BOOL;			// 長按已生效中,期間 LowCV 持續後退
	trigBTN_ShortPress	:BOOL;			// 短按事件 (放開且未進入長按)
	trigRequest		:R_TRIG;
	tonBtnCtrl		:ton;
	tonBtnMotorCtrl	:ton;
	tonBlinkTimer :TON;
	tonBlink_Internal :TIME :=T#500MS;

END_VAR

A00_BasicUnits();
SUPER^.A10_StateControl();

ACTION A00_BasicUnits:
tonBtnCtrl(PT:=T#5S);
tonBtnMotorCtrl(PT :=T#90S);
ErrorID := 2800;

// 長按 3s 觸發 NG 軌道(LowCV)後退;放開即停。短按沿用 (放開瞬間且 NOT bLongPressActive)。
ftrigBTN(CLK := Input.bStorage_StackPushPb);
trigBTN_ShortPress := ftrigBTN.Q AND NOT bLongPressActive;

tonLongPress(IN := Input.bStorage_StackPushPb, PT := T#3S);
IF tonLongPress.Q THEN
    bLongPressActive := TRUE;
END_IF

IF NOT Input.bStorage_StackPushPb AND bLongPressActive THEN
    Motor.List.LowCV.M_MotorStop();
    bLongPressActive := FALSE;
END_IF

IF bLongPressActive THEN
    Motor.List.LowCV.M_MoveBackward();
END_IF
END_ACTION

METHOD GetModelState
VAR_OUTPUT
    xDone    :BOOL;
    xBusy    :BOOL;
    xError   :BOOL;
    xAborted :BOOL;
    iErrorID :UDINT;
	UniqueErrorCode : STRING;
END_VAR
xDone    := Done;
xBusy    := Busy;
xError   := Error;
xAborted := Abort;
iErrorID := ErrorID;
END_METHOD

METHOD GetName : STRING
GetName := ObjectName;
END_METHOD

METHOD PRIVATE M_Blink : BOOL
VAR_INPUT
	
END_VAR
tonBlinkTimer(IN :=NOT tonBlinkTimer.Q,
				PT := tonBlink_Internal);
IF tonBlinkTimer.Q THEN
	Output.bStorage_StackPushPbLamp := NOT Output.bStorage_StackPushPbLamp;
END_IF
END_METHOD

METHOD PRIVATE M_GetCurrentStation : BOOL
VAR
	i : UINT;
	SetPos	 :LREAL;
END_VAR

VAR_OUTPUT
	uiCurrentStation	:UINT;
END_VAR
//SetPos := THIS^.fbMotor.NcToPlc.SetPos;
SetPos := arAxisCtrl_gb[AxisNo.RackMotor].Admin.Axis.NcToPlc.SetPos;
M_RefreshStationPos();
//IF  THIS^.fbMotor.Status.Homed THEN
IF arAxisCtrl_gb[AxisNo.RackMotor].Admin.Axis.Status.Homed THEN
	FOR i:=0 TO 9 BY 1 DO 
		IF SetPos> RackMotorStationTable[i].Position-5 AND SetPos< RackMotorStationTable[i].Position+5 THEN // Range should be confirm
			uiCurrentStation :=i;
			M_GetCurrentStation :=TRUE;
			RETURN;
		END_IF
	END_FOR
	
	uiCurrentStation:=99;
	M_GetCurrentStation :=FALSE;
ELSE
	M_GetCurrentStation :=FALSE;
	uiCurrentStation:=99;
END_IF
END_METHOD

METHOD PRIVATE M_MoveToStation : BOOL
VAR_INPUT
	uiStation : UINT;
END_VAR
VAR
	bDone	:BOOL;
	uiTargetPosition	:LREAL ;
END_VAR
M_RefreshStationPos();
IF uiStation>=0 AND uiStation <10 THEN
	uiTargetPosition :=RackMotorStationTable[uiStation].Position;
	
	arAxisCtrl_gb[AxisNo.RackMotor].PosMode.Acc := CurrentData.Axes.RackMotor.HalfAuto.Acceleration;
	arAxisCtrl_gb[AxisNo.RackMotor].PosMode.Dec := CurrentData.Axes.RackMotor.HalfAuto.Deceleration;
	arAxisCtrl_gb[AxisNo.RackMotor].PosMode.Jerk := CurrentData.Axes.RackMotor.HalfAuto.Jerk;
	arAxisCtrl_gb[AxisNo.RackMotor].PosMode.Velocity := CurrentData.Axes.RackMotor.HalfAuto.Velocity;
	arAxisCtrl_gb[AxisNo.RackMotor].PosMode.Position := uiTargetPosition;
	
//	THIS^.fbMotor.MoveAbs(lrPosition	:=uiTargetPosition,
//						lrVelocity 		:=GVL.MotorCore[AxisNo.RackMotor].VCC,
//						lrAcceleration	:=GVL.MotorCore[AxisNo.RackMotor].ACC,
//						lrDeceleration	:=GVL.MotorCore[AxisNo.RackMotor].DCC,
//						lrJerk			:=GVL.MotorCore[AxisNo.RackMotor].Jerk,
//						BufferMode		:=MC_BufferMode.MC_Aborting);
	//THIS^.fbMotor.GetCmdDoneStatus(bMotionCmdDone=>bDone);
ELSE
	M_MoveToStation :=FALSE;
	RETURN;
END_IF
END_METHOD

METHOD PRIVATE M_RefreshStationPos : BOOL
VAR_INPUT
END_VAR
VAR
	i: UINT;
	position : ST_PositionTable;
END_VAR
FOR i := 0 TO 9 DO
	position :=FUN_GetPositionTableData(PositionName:='W',Index:=i,Clip:=0);
RackMotorStationTable[i].Position:= position.X_Pos;
END_FOR
	M_RefreshStationPos :=TRUE;

// todo : update position of each stations
//FOR i:=1 TO 200 BY 1 DO
//	FOR iIndex:=0 TO 9 BY 1 DO
//		IF 		
//			DAS_CoreSys.MachineControl.CurrentData.PositionTable[i].Index= iIndex AND
//			DAS_CoreSys.MachineControl.CurrentData.PositionTable[i].Zone ='W' THEN
//			RackMotorStationTable[iIndex].Position := DAS_CoreSys.MachineControl.CurrentData.PositionTable[i].X_Pos;

//			StationsPosition[iIndex]:=RackMotorStationTable[i].Position;
//		ELSE
//			M_RefreshStationPos :=FALSE;
//		END_IF
//	END_FOR
//END_FOR
END_METHOD

METHOD  M_STATE_ABORTED
VAR_INPUT
END_VAR
ERROR :=TRUE;
Busy    := FALSE;
Aborted := TRUE;
Status := strStatus;

IF NOT Execute THEN
	eSTATE:=STATE_RESETTING;
END_IF

IF Execute AND Reset THEN
	uiExecutingStep :=uiResumeStep;
	eSTATE:=STATE_EXECUTING;
END_IF
END_METHOD

METHOD  M_STATE_ABORTING
VAR_INPUT
END_VAR
CASE uiAbortingStep OF
	0 :
		uiAbortingStep:=9999;
	
	9999:	_AbortCompleted:=TRUE;
END_CASE

IF _AbortCompleted THEN	
	eSTATE :=STATE_ABORTED;
END_IF
END_METHOD

METHOD  M_STATE_DONE
VAR_INPUT
END_VAR
Busy 	:= FALSE;
Done	:=TRUE;

IF NOT Execute THEN
	eSTATE:=STATE_RESETTING;
END_IF
END_METHOD

METHOD  M_STATE_DORMANT
VAR_INPUT
END_VAR
Busy            := FALSE;
Done            := FALSE;
Aborted         := FALSE;
Error           := FALSE;
ErrorID         := 0;
Status          := '';
_ResetCompleted := FALSE;
_Error          := FALSE;
_Executed       := FALSE;
strStatus :='FB_BoxSupplyCtrl_v1: No Error';
uiExecutingStep :=uiResettingStep :=uiResumeStep :=0;

IF Execute THEN
	eSTATE:=STATE_EXECUTING;
END_IF
END_METHOD

METHOD  M_STATE_ERROR
VAR_INPUT
END_VAR
ERROR   :=TRUE;
Busy	:=FALSE;
Status := strStatus;
M_TurnOff();
RackState:= E_RackState.idle; // Useless so far
AxisRackMotorBTNHomeRequest :=false;
IF NOT Execute OR Reset THEN // Execute will always on , therefor Reset is only way to recovery from error	
	eSTATE:=STATE_RESETTING;
END_IF
END_METHOD

METHOD  M_STATE_EXECUTING
VAR_INPUT
END_VAR

VAR_INST
	uiTransitingStep : UINT;
	uiTargetStation :UINT :=0;
	bFreeState	  :BOOL;
END_VAR

VAR
	bMotionDone			:BOOL;
	_uiCurrentStation	:UINT;
END_VAR
Busy :=TRUE;	
//IF SupplyBTN.P_IsBTNRef THEN			//2nd machine 
//	trigBTN(CLK:= (SupplyBTN.P_ButtonState));
//END_IF //Make sure BTN is referenced otherwise exception occur

	// trigBTN_ShortPress 由 A00_BasicUnits 中 ftrigBTN 計算 (放開瞬間且未進長按)
trigRequest(CLK :=(AddBoxes_Status.InterventionRequest AND bFreeState));

// Force state control
IF fbstorageHome.xDone THEN
	ExcutingStep := E_RackState.FeedBox;
	
ELSIF fbstorageHome.xBusy THEN
	ExcutingStep := E_RackState.ManualCtrl;
ELSIF AddBoxes_Status.Busy OR AddBoxes_Status.Done  AND NOT RackState = E_RackState.TransitingFeedBox THEN	
	ExcutingStep := E_RackState.AddBoxes;
	
ELSIF StroageRegionMode = E_UnitMode.MANUAL AND
	arAxisCtrl_gb[AxisNo.RackMotor].Admin.Axis.Status.HasJob AND
//	  rackmotor.fbMotor.Status.HasJob AND 
	  NOT (ExcutingStep = E_RackState.FeedBox)  AND 
		NOT (ExcutingStep = E_RackState.TransitingFeedBox) THEN	
			ExcutingStep := E_RackState.ManualCtrl;

ELSIF	StroageRegionMode = E_UnitMode.MANUAL AND 
		NOT Cylinder.List.fbStackPush.InRearPosition AND
//		BoxesPusherCylinder.P_IsMoving AND 
		NOT	(ExcutingStep = E_RackState.FeedBox) AND
		NOT (ExcutingStep = E_RackState.TransitingFeedBox)  THEN	
			ExcutingStep := E_RackState.ManualCtrl;

			
END_IF

RackState := ExcutingStep;

CASE ExcutingStep OF
	

	E_RackState.idle:
		;	
	E_RackState.AddBoxes:
		//Service AddBox working
		M_TurnOff();
		bFreeState:=FALSE;
		IF NOT AddBoxes_Ctrl.Execute AND NOT AddBoxes_Status.Error  THEN
        	ExcutingStep := E_RackState.Free;
    	END_IF
		
	E_RackState.ManualCtrl:
	//Stroage area in manual and Rack is moving
		M_TurnOff();
		bFreeState:=FALSE;
		IF NOT arAxisCtrl_gb[AxisNo.RackMotor].Admin.Axis.Status.HasJob AND Cylinder.List.fbStackPush.InRearPosition THEN
            ExcutingStep := E_RackState.Free;
        END_IF
		
	E_RackState.FeedBox:
	// FeedBox mode , 
		M_Blink();
		bFreeState:=FALSE;
		AxisRackMotorBTNHomeRequest :=false;
			IF	trigBTN_ShortPress THEN
				ExcutingStep :=E_RackState.TransitingFree;
			END_IF
			
	E_RackState.Free:
	// Rack is free , User is allow to ask to suply box by push the suplyBTN
		M_TurnOn();
		bFreeState:=TRUE;
			 IF trigBTN_ShortPress OR trigRequest.Q THEN
				 uiTransitingStep:=0;
				 ExcutingStep := E_RackState.TransitingFeedBox;
			 END_IF

	E_RackState.TransitingFree:
			 IF NOT AddBoxes_Status.InterventionRequest THEN
				 ExcutingStep :=E_RackState.Free;	
			 END_IF
		
	E_RackState.TransitingFeedBox:
	//Transition step , from Free to FeedBox
		//M_Blink();
		M_TurnOff();
		bFreeState:=FALSE;
		AxisRackMotorBTNHomeRequest :=TRUE;
		// todo : if transition step needs different indication of BTN behavior?
		CASE uiTransitingStep OF
		0:
			tonBtnCtrl.IN	:=FALSE;
			tonBtnMotorCtrl.IN :=FALSE;
			uiTransitingStep:=5;
			M_GetCurrentStation(uiCurrentStation =>_uiCurrentStation);
			IF uiTargetStation = _uiCurrentStation THEN
				uiTransitingStep :=30;
			END_IF
			
		5:	//Move cylinder back
			tonBtnCtrl.IN:=TRUE;			
			Cylinder.List.fbStackPush.M_Retract();
			IF Cylinder.List.fbStackPush.InRearPosition AND NOT arAxisCtrl_gb[AxisNo.RackMotor].Admin.Axis.Status.HasJob THEN 
				tonBtnCtrl.IN :=FALSE;
				uiTransitingStep :=10;
			END_IF
			IF tonBtnCtrl.Q THEN
				_Error:= TRUE;
				StrStatus :='FB_BoxSupplyCtrl_v1 Step 5: Cylinder MoveBackward timeout';
			END_IF
		10:	// Rackmotor move to station 0
			tonBtnMotorCtrl.IN :=TRUE;
			M_MoveToStation(uiTargetStation);
			IF arAxisCtrl_gb[AxisNo.RackMotor].Admin.Axis.Status.HasJob THEN
			uiTransitingStep :=20;
			END_IF
			IF tonBtnMotorCtrl.Q THEN
				_Error :=TRUE;
				StrStatus :='FB_BoxSupplyCtrl_v1 Step 10: RackMotor MoveToStation timeout';
			END_IF
		20:	// check currentstation 
			tonBtnMotorCtrl.IN :=TRUE;
//			bMotionDone :=rackmotor.fbMotor.Status.InTargetPosition;
			bMotionDone :=arAxisCtrl_gb[AxisNo.RackMotor].Admin.Axis.Status.InTargetPosition;
			M_GetCurrentStation(uiCurrentStation =>_uiCurrentStation);
			IF bMotionDone  AND uiTargetStation = _uiCurrentStation THEN
				tonBtnMotorCtrl.IN :=FALSE;
				uiTransitingStep :=30;
			END_IF
			IF tonBtnMotorCtrl.Q THEN
				_Error :=TRUE;
				StrStatus :='FB_BoxSupplyCtrl_v1 Step 20: RackMotor currentStation timeout';
			END_IF
		30:
			ExcutingStep := E_RackState.FeedBox;
			AxisRackMotorBTNHomeRequest :=FALSE;
		END_CASE
		


END_CASE
	
IF NOT Execute THEN
	eState:=STATE_RESETTING;
END_IF
IF _Error THEN
	eState:=STATE_ERROR;
END_IF
IF _Abort THEN
	eSTATE:=STATE_ABORTING;
END_IF
IF _Executed THEN
	eSTATE:=STATE_Done;
END_IF
END_METHOD

METHOD  M_STATE_RESETTING
VAR_INPUT
END_VAR
Error :=FALSE;
Done :=FALSE;
Busy := FALSE;
AxisRackMotorBTNHomeRequest :=FALSE;
tonBtnCtrl.IN := FALSE;
tonBtnMotorCtrl.IN := FALSE;
M_TurnOff();
CASE uiResettingStep OF
	
	0:
		uiResettingStep:=9999;


	9999:
		_ResetCompleted:=TRUE;
END_CASE
IF _ResetCompleted THEN
	eSTATE:=STATE_DORMANT;
END_IF
END_METHOD

METHOD PRIVATE M_TurnOff : BOOL
VAR_INPUT
END_VAR
Output.bStorage_StackPushPbLamp := false;
END_METHOD

METHOD PRIVATE M_TurnOn : BOOL
VAR_INPUT
END_VAR
Output.bStorage_StackPushPbLamp := true;
END_METHOD

END_FUNCTION_BLOCK

// ---- Library/20_MachineUnits/21_StorageArea/Service/FB_RebootModbusDevice.TcPOU
FUNCTION_BLOCK FB_RebootModbusDevice EXTENDS FB_ActionBasic
VAR_INPUT
	xExecute : BOOL;
	xAbort : BOOL;  
	OutPut           : REFERENCE TO ST_OutputTable;
	OffDelayTime	 : INT ; // in second //default 2 s if C# no assign
	OnDelayTime		 : INT ; // in second
END_VAR
VAR_OUTPUT
	xAborted : BOOL;
	iErrorID : INT;
	ErrorMsg : T_MaxString;

END_VAR
VAR
	StateBehaviour : CBML.ETrigA;		
	uiModBusStep : UINT :=0;
	tonDelay	 : TON;
END_VAR

THIS^.IBehaviourModel := StateBehaviour;
StateBehaviour(xExecute := xExecute,
    xDone => xDone,
    xBusy => xBusy,
    xError => xError,
    xAbort := xAbort,
    xAborted => xAborted);

iErrorID := StateBehaviour._model.iErrorID;
ErrorMsg := M_GetErrorMsg(xErrorID := iErrorID);
tonDelay();

METHOD CleanupAction
VAR_INPUT
    xAbortProposed : BOOL;
    iErrorIDProposed: INT;
END_VAR
VAR_OUTPUT
    xComplete : BOOL := TRUE;
    xAbort: BOOL := xAbortProposed;
 	iErrorID : INT := iErrorIDProposed;
END_VAR
END_METHOD

METHOD CyclicAction
VAR_INPUT
    itfTimingController : CBML.ITimingController;
END_VAR
VAR_OUTPUT
    xComplete : BOOL := TRUE;
    iErrorID : INT := 0;
END_VAR
VAR
	DelayTime : TIME;
END_VAR
xComplete := FALSE;


CASE uiModBusStep OF
		0:// Switch off RS485 power 
			
			OutPut.bTurnOffRS485Sensors_1 := TRUE;
			OutPut.bTurnOffRS485Sensors_2 := TRUE;
			GVL_Machine.stModbusByPassInternal.switchOff_1 := TRUE;
			GVL_Machine.stModbusByPassInternal.switchOff_2 := TRUE;
			GVL_Machine.stModbusByPassInternal.switchOff_3 := TRUE;
			GVL_Machine.stModbusByPassInternal.switchOff_4 := TRUE;
			DelayTime := INT_TO_TIME(OffDelayTime) *1000;	
			tonDelay.PT:=DelayTime;
			//tonDelay.IN :=TRUE;
			uiModBusStep:=100;
		100:
			tonDelay.IN :=TRUE;
			IF 	tonDelay.Q THEN
				uiModBusStep:=200;
			END_IF
		200:// Power on again
			OutPut.bTurnOffRS485Sensors_1 := FALSE	;
			OutPut.bTurnOffRS485Sensors_2 := FALSE;
			tonDelay.IN :=FALSE;
			IF NOT 	tonDelay.Q THEN
				uiModBusStep:=300;
			END_IF
		300: // Wait another time make sure modules boot
			DelayTime := INT_TO_TIME(OffDelayTime) *1000;	
			tonDelay.PT:=DelayTime;
			tonDelay.IN :=TRUE;	
			IF 	tonDelay.Q THEN
				uiModBusStep:=400;
			END_IF
		400:
			tonDelay.IN :=FALSE;
			uiModBusStep :=500;
			
			
		500://Step done	
			DelayTime := INT_TO_TIME(OffDelayTime) *1000;			//delay on ModBus Service edit by min 20250927
			tonDelay.PT:=DelayTime;
			tonDelay.IN :=TRUE;
			IF tonDelay.Q THEN
			GVL_Machine.stModbusByPassInternal.switchOff_1 := FALSE;
			GVL_Machine.stModbusByPassInternal.switchOff_2 := FALSE;
			GVL_Machine.stModbusByPassInternal.switchOff_3 := FALSE;
			GVL_Machine.stModbusByPassInternal.switchOff_4 := FALSE;
			uiModBusStep:=9000;
			END_IF
		9000:
			xComplete := TRUE;	
END_CASE
END_METHOD

METHOD ExitAction
VAR_INPUT
    xAfterCleanup : BOOL;
    xInCopyCode : BOOL;
END_VAR
uiModBusStep := 0;
END_METHOD

METHOD M_GetErrorMsg : T_MaxString
VAR_INPUT
	xErrorID: INT;
END_VAR

VAR
	
END_VAR
CASE xErrorID OF
    0:
        M_GetErrorMsg := 'No Error';
    1:
        M_GetErrorMsg := 'FB_RebootModbusDevice ErrorID 1: Action time out';
    2:
        M_GetErrorMsg := 'FB_RebootModbusDevice ErrorID 2: Cylinder not ready';
    3:
        M_GetErrorMsg := 'FB_RebootModbusDevice ErrorID 3: Motor not ready';
    4:
		M_GetErrorMsg := 'FB_RebootModbusDevice ErrorID 4: FanucRobot can not homing';
END_CASE
END_METHOD

METHOD ResetAction
VAR_OUTPUT
    xComplete : BOOL := TRUE;
END_VAR
OutPut.bTurnOffRS485Sensors_1 := FALSE;
OutPut.bTurnOffRS485Sensors_2 := FALSE;
GVL_Machine.stModbusByPassInternal.switchOff_1 := FALSE;
GVL_Machine.stModbusByPassInternal.switchOff_2 := FALSE;
GVL_Machine.stModbusByPassInternal.switchOff_3 := FALSE;
GVL_Machine.stModbusByPassInternal.switchOff_4 := FALSE;
uiModBusStep:=0;
tonDelay.IN := FALSE;
END_METHOD

METHOD StartAction
VAR_OUTPUT
    xComplete : BOOL := TRUE;
	iErrorID : INT := 0;
END_VAR

VAR
	uiCylinderIndex :UINT;
	uiMotorIndex : UINT;
END_VAR
GVL_Machine.stModbusByPassInternal.switchOff_1 := FALSE;
GVL_Machine.stModbusByPassInternal.switchOff_2 := FALSE;
GVL_Machine.stModbusByPassInternal.switchOff_3 := FALSE;
GVL_Machine.stModbusByPassInternal.switchOff_4 := FALSE;
tonDelay.IN := FALSE;
uiModBusStep:=0;
END_METHOD

END_FUNCTION_BLOCK

// ---- Library/20_MachineUnits/23_ShippingArea/FB_ShippingArea.TcPOU
FUNCTION_BLOCK FB_ShippingArea EXTENDS FB_ModeBase_V2 IMPLEMENTS I_UnitState
VAR_INPUT
	FanucRobot 		: REFERENCE TO FB_FanucRobot_Basic_V2;
	Service 		: REFERENCE TO ST_ShippingService;
	INPUT       	: REFERENCE TO ST_InputTable;
	OUTPUT			: REFERENCE TO ST_OutputTable;
	Motor    		: REFERENCE TO UNI_MotorList;
	Cylinder		: REFERENCE TO UNI_CylinderList;
	SameSizeCVRequest : REFERENCE TO ST_SameSizeCVRequest;	// Phase 2 仲裁,傳到 fbShippingRobotTransfer / fbShippingPlateScan
	SameSizeCV_Press1_AlreadyExtended : REFERENCE TO BOOL;	// 一次性 latch (傳給 fbShippingPlateScan):首次 Scan 觸發 Press1 伸出後固定 TRUE
	SameSizeCV_Press3_AlreadyExtended : REFERENCE TO BOOL;	// 一次性 latch (傳給 fbShippingPlateScan):首次 Scan 觸發 Press3 伸出後固定 TRUE
    Reset           : REFERENCE TO BOOL;
	Stop 			: REFERENCE TO BOOL;
    bStopMem 		: REFERENCE TO BOOL;
END_VAR
VAR_OUTPUT
	Homed : BOOL;
	RobotResetCMD : BOOL;
END_VAR
VAR
	abort	: BOOL;

	// 連動暫停 - 任一 Service 錯誤時暫停所有其他 Service
	_bAnyServiceError : BOOL;

	//Machine Service
	fbShippingHoming 				: FB_ShippingHoming;
	
	// Same / Difference CV Service
	fbShippingRobot_TransmitCVEnd :	FB_ShippingRobot_TransmitCVEnd;

	//Robot Service
	fbShippingRobot_Left 			: FB_ShippingRobot_Left;
	fbShippingRobot_Right 			: FB_ShippingRobot_Right;
	fbShippingRobot_Buffer			: FB_ShippingRobot_Buffer;
	fbShippingRobot_PhotoStandByPos	: FB_ShippingRobot_PhotoStandByPos;
	fbShippingRobotTransfer			: FB_ShippingRobotTransfer;
	fbShippingPlateScan				: FB_ShippingPlateScan;

	//HansLaser HandShake TransCV Service
	fbShippingLeftSideTransCV		: FB_ShippingTransCV_LeftSide;
	fbShippingRightSideTransCV		: FB_ShippingTransCV_RightSide;
END_VAR

SUPER^();

IF __ISVALIDREF(PackTag) THEN
    eModeCommand  := PackTag.Command.UnitMode;
    eStateCommand := PackTag.Command.CntrlCmd;
ELSE
    RETURN;
END_IF

ACTION A00_Service:
// ============================================================================
// 連動暫停邏輯 - 任一 Service 錯誤時，暫停所有其他 Service
// ============================================================================
_bAnyServiceError := false;
//	Service.AutoMode_ShippingRobot_TransmitCVEnd.Status.Error OR
//	Service.AutoMode_ShippingRobot_Left.Status.Error OR
//	Service.AutoMode_ShippingRobot_Right.Status.Error OR
//	Service.AutoMode_ShippingTransCV_LeftSide.Status.Error OR
//	Service.AutoMode_ShippingTransCV_RightSide.Status.Error;

fbShippingRobot_TransmitCVEnd(
	Execute:= Service.AutoMode_ShippingRobot_TransmitCVEnd.Command.Execute,
	Abort:= Service.AutoMode_ShippingRobot_TransmitCVEnd.Command.Abort OR THIS^.Abort OR _bAnyServiceError,
	Reset:= Reset OR Service.AutoMode_ShippingRobot_TransmitCVEnd.Command.Reset, 
	ObjectName:= 'Shipping Fanuc Robot TransmitCVEnd', 
	INPUT:=INPUT,
	Motor :=Motor,
	Busy=> Service.AutoMode_ShippingRobot_TransmitCVEnd.Status.Busy, 
	Done=> Service.AutoMode_ShippingRobot_TransmitCVEnd.Status.Done, 
	Aborted=> , 
	Error=> Service.AutoMode_ShippingRobot_TransmitCVEnd.Status.Error, 
	ErrorID=> , 
	Status=> Service.AutoMode_ShippingRobot_TransmitCVEnd.Status.Status, 
	UniqueErrorCode=> , 
	Robot:= FanucRobot, 
	Info:= Service.AutoMode_ShippingRobot_TransmitCVEnd.Info, 
	Stop:= bStopMem,
	fbSHippingHomingBusy := fbShippingHoming.xBusy);
	
fbShippingRobot_Left(
	Execute:= service.AutoMode_ShippingRobot_Left.Command.Execute,
	Abort:= Service.AutoMode_ShippingRobot_Left.Command.Abort OR THIS^.Abort OR _bAnyServiceError,
	Reset:= Reset OR Service.AutoMode_ShippingRobot_Left.Command.Reset,
	ObjectName:= 'Shipping Fanuc Robot Left', 
	Busy=> Service.AutoMode_ShippingRobot_Left.Status.Busy, 
	Done=> Service.AutoMode_ShippingRobot_Left.Status.Done, 
	Aborted=> , 
	Error=> Service.AutoMode_ShippingRobot_Left.Status.Error, 
	ErrorID=> , 
	Status=> Service.AutoMode_ShippingRobot_Left.Status.Status, 
	UniqueErrorCode=> , 
	Robot:= FanucRobot, 
	Info:= Service.AutoMode_ShippingRobot_Left.Info, 
	Stop:=bStopMem,
	Buzz := DAS_CoreSys.MachineControl._Buzz,
	RedLamp:= DAS_CoreSys.MachineControl._RedLamp,
	bCompleteRequest := Service.AutoMode_ShippingRobot_Left.bCompleteRequest,
	bTransCVInPosition => Service.AutoMode_ShippingRobot_Left.bTransCVInPosition,
	Input := INPUT);
	
fbShippingRobot_Right(
	Execute:= Service.AutoMode_ShippingRobot_Right.Command.Execute,
	Abort:= Service.AutoMode_ShippingRobot_Right.Command.Abort OR THIS^.Abort OR _bAnyServiceError,
	Reset:= Reset OR Service.AutoMode_ShippingRobot_Right.Command.Reset,
	ObjectName:= 'Shipping Fanuc Robot Right', 
	Busy=> Service.AutoMode_ShippingRobot_Right.Status.Busy, 
	Done=> Service.AutoMode_ShippingRobot_Right.Status.Done, 
	Aborted=> , 
	Error=> Service.AutoMode_ShippingRobot_Right.Status.Error, 
	ErrorID=> , 
	Status=> Service.AutoMode_ShippingRobot_Right.Status.Status, 
	UniqueErrorCode=> , 
	Robot:= FanucRobot, 
	Info:= Service.AutoMode_ShippingRobot_Right.Info, 
	Stop:= bStopMem,
	Buzz := DAS_CoreSys.MachineControl._Buzz,
	RedLamp:= DAS_CoreSys.MachineControl._RedLamp,
	bCompleteRequest := Service.AutoMode_ShippingRobot_Right.bCompleteRequest,
	bTransCVInPosition => Service.AutoMode_ShippingRobot_Right.bTransCVInPosition,
	Input := INPUT);
	
fbShippingHoming(
	xDone=> ,
	xBusy=> ,
	xError=> ,
	xExecute:= ,
	xAbort:= _bAnyServiceError,
	FanucRobot:= FanucRobot, 
	Homed:= Homed, 
	xAborted=> , 
	iErrorID=> , 
	ErrorMsg=> , 
	RobotResetCMD=> RobotResetCMD,
	Service := Service,
	input := INPUT,
	Output := OUTPUT,
	Motor := Motor);
	
fbShippingLeftSideTransCV(
	xDone=> Service.AutoMode_ShippingTransCV_LeftSide.Status.Done,
	xBusy=> Service.AutoMode_ShippingTransCV_LeftSide.Status.Busy,
	xError=> Service.AutoMode_ShippingTransCV_LeftSide.Status.Error,
	xExecute:= Service.AutoMode_ShippingTransCV_LeftSide.Command.Execute,
	xAbort:= Service.AutoMode_ShippingTransCV_LeftSide.Command.Abort OR THIS^.abort OR _bAnyServiceError,
	xReset:= Service.AutoMode_ShippingTransCV_LeftSide.Command.Reset,
	Cylinder:= , 
	TimeOut:= , 
	Input:= input, 
	OutPut:= output, 
	Motor:= , 
	ShippingTransCVRequest_LeftSide:= Service.AutoMode_ShippingTransCV_LeftSide.ShippingTransCVRequest_LeftSide, 
	RobotStatus:= Service.AutoMode_ShippingRobot_Left.Status, 
	xAborted=> , 
	iErrorID=> , 
	ErrorMsg=> Service.AutoMode_ShippingTransCV_LeftSide.Status.Status);
	
fbShippingRightSideTransCV(
	xDone=> Service.AutoMode_ShippingTransCV_RightSide.Status.Done,
	xBusy=> Service.AutoMode_ShippingTransCV_RightSide.Status.Busy,
	xError=> Service.AutoMode_ShippingTransCV_RightSide.Status.Error,
	xExecute:= Service.AutoMode_ShippingTransCV_RightSide.Command.Execute,
	xAbort:= Service.AutoMode_ShippingTransCV_RightSide.Command.Abort OR THIS^.abort OR _bAnyServiceError,
	xReset:= Service.AutoMode_ShippingTransCV_RightSide.Command.Reset,
	Cylinder:= , 
	TimeOut:= , 
	Input:= input, 
	OutPut:= output, 
	Motor:= , 
	ShippingTransCVRequest_RightSide:= Service.AutoMode_ShippingTransCV_RightSide.ShippingTransCVRequest_RightSide, 
	RobotStatus:= Service.AutoMode_ShippingRobot_Right.Status, 
	xAborted=> , 
	iErrorID=> , 
	ErrorMsg=> Service.AutoMode_ShippingTransCV_RightSide.Status.Status);


fbShippingRobotTransfer(
	Execute:= Service.AutoMode_ShippingRobotTransfer.Command.Execute,
	Abort:= Service.AutoMode_ShippingRobotTransfer.Command.Abort OR THIS^.Abort OR _bAnyServiceError,
	Reset:= Reset OR Service.AutoMode_ShippingRobotTransfer.Command.Reset,
	Pause:= bStopMem,
	ObjectName:= 'FB_ShippingRobotTransfer',
	Busy=> Service.AutoMode_ShippingRobotTransfer.Status.Busy,
	Done=> Service.AutoMode_ShippingRobotTransfer.Status.Done,
	Aborted=> ,
	Error=> Service.AutoMode_ShippingRobotTransfer.Status.Error,
	Paused=> ,
	ErrorID=> ,
	Status=> Service.AutoMode_ShippingRobotTransfer.Status.Status,
	UniqueErrorCode=> ,
	Robot:= FanucRobot,
	Info:= Service.AutoMode_ShippingRobotTransfer.Info,
	Stop:= bStopMem,
	Input:= INPUT,
	Output:= OUTPUT,
	Motor:= Motor,
	SameSizeCVRequest:= SameSizeCVRequest,
	Cylinder:= Cylinder,
	Buzz:= DAS_CoreSys.MachineControl._Buzz,
	RedLamp:= DAS_CoreSys.MachineControl._RedLamp,
	bCompleteRequest:= Service.AutoMode_ShippingRobotTransfer.bCompleteRequest,
	bTransCVInPosition_Left=> Service.AutoMode_ShippingRobotTransfer.bTransCVInPosition_Left,
	bTransCVInPosition_Right=> Service.AutoMode_ShippingRobotTransfer.bTransCVInPosition_Right,
	fbShippingHomingBusy:= fbShippingHoming.xBusy);
	
fbShippingRobot_Buffer(
	Execute:= Service.AutoMode_ShippingRobot_Buffer.Command.Execute, 
	Abort:= Service.AutoMode_ShippingRobot_Buffer.Command.Abort, 
	Reset:= Service.AutoMode_ShippingRobot_Buffer.Command.Reset, 
	Pause:= bStopMem, 
	ObjectName:= 'FB_ShippingRobot_Buffer', 
	Busy=> Service.AutoMode_ShippingRobot_Buffer.Status.Busy, 
	Done=> Service.AutoMode_ShippingRobot_Buffer.Status.Done, 
	Aborted=> , 
	Error=> Service.AutoMode_ShippingRobot_Buffer.Status.Error, 
	Paused=> , 
	ErrorID=> , 
	Status=> Service.AutoMode_ShippingRobot_Buffer.Status.Status, 
	UniqueErrorCode=> , 
	Robot:= fanucrobot, 
	Info:= Service.AutoMode_ShippingRobot_Buffer.Info, 
	Stop:= , 
	Input:= INPUT, 
	Output:= OUTPUT,
	Cylinder := cylinder);
	
fbShippingRobot_PhotoStandByPos(
	Execute:= Service.AutoMode_ShippingRobot_PhotoStandByPos.Command.Execute, 
	Abort:= Service.AutoMode_ShippingRobot_PhotoStandByPos.Command.Abort, 
	Reset:=  Service.AutoMode_ShippingRobot_PhotoStandByPos.Command.Reset, 
	Pause:= bStopMem, 
	ObjectName:= 'FB_ShippingRobot_PhotoStandByPos', 
	Busy=> Service.AutoMode_ShippingRobot_PhotoStandByPos.Status.Busy, 
	Done=> Service.AutoMode_ShippingRobot_PhotoStandByPos.Status.Done, 
	Aborted=> , 
	Error=> Service.AutoMode_ShippingRobot_PhotoStandByPos.Status.Error, 
	Paused=> , 
	ErrorID=> , 
	Status=> Service.AutoMode_ShippingRobot_PhotoStandByPos.Status.Status, 
	UniqueErrorCode=> ,
	Robot:= ,
	Info:= Service.AutoMode_ShippingRobot_PhotoStandByPos.Info,
	Stop:= ,
	Input:= INPUT,
	Output:= OUTPUT);

fbShippingPlateScan(
	Execute:= Service.AutoMode_ShippingPlateScan.Command.Execute,
	Abort:= Service.AutoMode_ShippingPlateScan.Command.Abort OR THIS^.Abort OR _bAnyServiceError,
	Reset:= Reset OR Service.AutoMode_ShippingPlateScan.Command.Reset,
	Pause:= bStopMem,
	ObjectName:= 'FB_ShippingPlateScan',
	Busy=> Service.AutoMode_ShippingPlateScan.Status.Busy,
	Done=> Service.AutoMode_ShippingPlateScan.Status.Done,
	Aborted=> ,
	Error=> Service.AutoMode_ShippingPlateScan.Status.Error,
	Paused=> ,
	ErrorID=> ,
	Status=> Service.AutoMode_ShippingPlateScan.Status.Status,
	UniqueErrorCode=> ,
	Robot:= FanucRobot,
	Motor:= Motor,
	SameSizeCVRequest:= SameSizeCVRequest,
	Cylinder:= Cylinder,
	SameSizeCV_Press1_AlreadyExtended:= SameSizeCV_Press1_AlreadyExtended,
	SameSizeCV_Press3_AlreadyExtended:= SameSizeCV_Press3_AlreadyExtended,
	Input:= INPUT,
	Side:= Service.AutoMode_ShippingPlateScan.Side,
	PlateIndex:= Service.AutoMode_ShippingPlateScan.PlateIndex,
	ReadComplete:= Service.AutoMode_ShippingPlateScan.ReadComplete,
	PlateHasBox=> Service.AutoMode_ShippingPlateScan.PlateHasBox,
	FeedBack=> Service.AutoMode_ShippingPlateScan.FeedBack);
END_ACTION

METHOD M_Aborted
abort := false;
M_StateComplete();
END_METHOD

METHOD M_Aborting
abort := true;
M_StateComplete();
END_METHOD

METHOD M_Clearing
M_StateComplete();
END_METHOD

METHOD M_Complete
M_StateComplete();
END_METHOD

METHOD M_Completing
M_StateComplete();
END_METHOD

METHOD M_Execute
CASE eModeCurrent OF
	E_UnitMode.Manual:
		;
	E_UnitMode.Auto:
		;
END_CASE
A00_Service();
//M_StateComplete();
END_METHOD

METHOD M_Held
M_StateComplete();
END_METHOD

METHOD M_Holding
M_StateComplete();
END_METHOD

METHOD M_Idle
M_StateComplete();
END_METHOD

METHOD M_Resetting
M_StateComplete();
END_METHOD

METHOD M_StartHoming
VAR_INPUT
END_VAR
fbShippingHoming.xExecute := TRUE;
END_METHOD

METHOD M_Starting
M_StateComplete();
END_METHOD

METHOD M_StopHoming
VAR_INPUT
END_VAR
fbShippingHoming.xExecute := False;
END_METHOD

METHOD M_Stopped
M_StateComplete();
END_METHOD

METHOD M_Stopping
M_StateComplete();
END_METHOD

METHOD M_Suspended
M_StateComplete();
END_METHOD

METHOD M_Suspending
M_StateComplete();
END_METHOD

METHOD M_Undefined
M_StateComplete();
END_METHOD

METHOD M_Unholding
M_StateComplete();
END_METHOD

METHOD M_Unsuspending
M_StateComplete();
END_METHOD

END_FUNCTION_BLOCK

// ---- Library/20_MachineUnits/23_ShippingArea/FB_ShippingHoming.TcPOU
FUNCTION_BLOCK FB_ShippingHoming EXTENDS FB_ActionBasic
VAR_INPUT
	xExecute 	: BOOL;
	xAbort 		: BOOL;
    FanucRobot 	: REFERENCE TO FB_FanucRobot_Basic_V2;
	Homed 		: REFERENCE TO BOOL;
	input		: REFERENCE TO ST_InputTable;
	Output		: REFERENCE TO ST_OutputTable;
	Service		: REFERENCE TO ST_ShippingService;
	Motor		: REFERENCE TO UNI_MotorList;
END_VAR
VAR_OUTPUT
	xAborted : BOOL;
	iErrorID : INT;
	ErrorMsg : STRING;
	RobotResetCMD : BOOL;
END_VAR
VAR
	StateBehaviour 		 : CBML.ETrigA;
	uiShippingHomingStep : UINT;
	FanucRobotCheckTon 	 	: TON;
	ResetRobotDelay 	 	: TON;
	TON_RobotFeedOutCommand : TON;
	TON_RobotTimeOut		: TON;
	fbExecuteEdgeDetect  :FB_EdgeDetect;
	_fbShippingRobot_TransmitCVEnd	: FB_ShippingRobot_TransmitCVEnd;
	TON_RobotRSR01_Delay	: TON;
	
	//Reboot RobotPower
	TON_RebootPowerDelay	: TON;
	TON_ConnectionTimeout	: TON;

	// 啟動延時 - 等待心跳偵測完成 (冷啟動用)
	TON_StartupDelay		: TON;
END_VAR

A00_BasicUnits();
THIS^.IBehaviourModel := StateBehaviour;
StateBehaviour(xExecute := xExecute,
    xDone => xDone,
    xBusy => xBusy,
    xError => xError,
    xAbort := xAbort OR fbExecuteEdgeDetect.xFallingEdge,
    xAborted => xAborted);

//Error Msg
iErrorID := StateBehaviour._model.iErrorID;
ErrorMsg := M_GetErrorMsg(xErrorID := iErrorID);


//Make sure that C# turns off execute to shut down the service
fbExecuteEdgeDetect(xInput :=xExecute);

ACTION A00_BasicUnits:
FanucRobotCheckTon(PT := T#90S);		//All Service TimeOut
ResetRobotDelay(PT:=T#300MS);
TON_RobotFeedOutCommand(PT:= T#5S);		//Robot FeedOut Command TimeOut
TON_RobotTimeOut(PT := T#60S);			//Robot FeedOut Service Done Time
TON_RobotRSR01_Delay(PT :=T#3S);
TON_RebootPowerDelay(PT :=T#5S);		// 電源 TRUE 維持 5 秒 (與大手臂同步，避免 24V 電容殘電造成假性斷電)
TON_ConnectionTimeout(PT :=T#60S);
TON_StartupDelay(PT :=T#5S);			// 啟動延時 5 秒 (等待心跳偵測冷啟動完成)


_fbShippingRobot_TransmitCVEnd(
	Execute:= , 
	Abort:= , 
	Reset:= , 
	ObjectName:= , 
	Busy=> , 
	Done=> , 
	Aborted=> , 
	Error=> , 
	ErrorID=> , 
	Status=> , 
	UniqueErrorCode=> , 
	Robot:= fanucrobot, 
	Info:= , 
	Stop:= , 
	INPUT:= input, 
	Motor:= Motor, 
	bCompleteRequest:= ,
	fbSHippingHomingBusy := THIS^.xBusy);
END_ACTION

METHOD CleanupAction
VAR_INPUT
    xAbortProposed : BOOL;
    iErrorIDProposed: INT;
END_VAR
VAR_OUTPUT
    xComplete : BOOL := TRUE;
    xAbort: BOOL := xAbortProposed;
 	iErrorID : INT := iErrorIDProposed;
END_VAR
RobotResetCMD := FALSE;
FanucRobotCheckTon.IN := FALSE;
uiShippingHomingStep := 0;
END_METHOD

METHOD CyclicAction
VAR_INPUT
    itfTimingController : CBML.ITimingController;
END_VAR
VAR_OUTPUT
    xComplete : BOOL := TRUE;
    iErrorID : INT := 0;
END_VAR
xComplete := FALSE;
CASE uiShippingHomingStep OF
	
	0:		//init
			TON_RobotFeedOutCommand.IN  := FALSE;
			TON_RobotTimeOut.IN 		:= FALSE;
			FanucRobotCheckTon.IN 		:= TRUE;
			uiShippingHomingStep 	    := 5;

	// ============================================================================
	// Step 5: 啟動延時 - 等待心跳偵測完成
	// - 冷啟動時，心跳偵測需要 5 秒 (10 × 0.5s) 才能判定連線狀態
	// - 必須等心跳偵測完成後，才能正確判斷機器人是否已連線，避免誤觸發電源循環
	// ============================================================================
	5:
			TON_StartupDelay.IN := TRUE;
			IF TON_StartupDelay.Q THEN
				TON_StartupDelay.IN := FALSE;
				uiShippingHomingStep := 10;
			END_IF

	10:		// 檢查機械手臂 錯誤狀態
			// 斷線判定: EIP scanner 報斷線 OR 軟體心跳 5 秒未翻轉 (iTestCnt >= 10)
			IF fanucrobot._EIPConnectionState = 8195 OR fanucrobot.iTestCnt >= 10 THEN
				FanucRobotCheckTon.IN := FALSE;					// 暫停 90 秒總超時，避免電源循環中誤觸發
				Output.bShipping_FanucRobotPower := TRUE;
				uiShippingHomingStep := 20;
			ELSIF fanucrobot.Halt THEN
				// Robot 在 Halt 狀態 → 清除 Hold 讓 Halt 解除，再 Reset 回 DORMANT
				fanucrobot.Hold := FALSE;
				fanucrobot.Reset := TRUE;
				ResetRobotDelay.IN := TRUE;
			ELSIF fanucrobot.Error THEN
				uiShippingHomingStep := 50;
			ELSIF fanucrobot._UO1.UO03_PrgRunning THEN
				// Robot 正在執行流程 → 強制停止後再切 RSR02
				fanucrobot.M_ResetAllCommand();
				fanucrobot.Hold := FALSE;
				fanucrobot.Reset := TRUE;
				ResetRobotDelay.IN := TRUE;
			ELSE
				uiShippingHomingStep := 500;
			END_IF
			IF ResetRobotDelay.Q THEN
				ResetRobotDelay.IN := FALSE;
				fanucrobot.Reset := FALSE;
				uiShippingHomingStep := 500;
			END_IF

	20:		// 電源 TRUE 維持 5 秒後切回 FALSE 重啟小手臂
			TON_RebootPowerDelay.IN :=TRUE;
			IF TON_RebootPowerDelay.Q THEN
				Output.bShipping_FanucRobotPower := FALSE;
				uiShippingHomingStep := 30;
			END_IF

	30:
			TON_RebootPowerDelay.IN  := FALSE;
			TON_ConnectionTimeout.IN := TRUE;
			IF TON_ConnectionTimeout.Q THEN
				// 超時 60 秒，連線失敗
				TON_ConnectionTimeout.IN := FALSE;
				iErrorID := 30;
				uiShippingHomingStep := 9999;
			ELSIF fanucrobot._EIPConnectionState <> 8195 AND fanucrobot.iTestCnt < 10 THEN
				// EIP 已重連 + 心跳已恢復，繼續檢查錯誤
				TON_ConnectionTimeout.IN := FALSE;
				FanucRobotCheckTon.IN := TRUE;					// 恢復 90 秒總超時監控
				uiShippingHomingStep := 50;
			END_IF
	
	50:
			IF FanucRobot.Error THEN
				RobotResetCMD := TRUE;
				ResetRobotDelay.IN:=TRUE;
			ELSE
				uiShippingHomingStep := 500;
			END_IF
			IF ResetRobotDelay.Q THEN
				ResetRobotDelay.IN :=FALSE;
				uiShippingHomingStep := 500;
			END_IF
		
		
	500:	// 手臂 RSR02 回原點
			ResetRobotDelay.IN := FALSE;
			RobotResetCMD := FALSE;
			FanucRobot.OpMode := E_FanucRobotOpMode.RSR02;
			IF FanucRobot.Error THEN
				RobotResetCMD := TRUE;		
			END_IF
			IF FanucRobot._RSR2_Completed THEN
				uiShippingHomingStep := 600;
			END_IF
			
	600:	// 回完回點後切換為 RSR01 工作模式
			FanucRobot.OpMode := E_FanucRobotOpMode.RSR01;
			IF FanucRobot._RSR1_Ready THEN
				uiShippingHomingStep := 1000;
			END_IF
			// RSR02 完成後，檢查是否還有殘留錯誤
			IF FanucRobot.Error THEN
				iErrorID := 21;		// RSR02 完成但錯誤仍存在
			END_IF
		
	1000:	// 確認手臂切換到 RSR01 模式，並且確保已回報 PLC 正在執行 RSR01
			IF FanucRobot.OpMode = E_FanucRobotOpMode.RSR01 AND 
				NOT FanucRobot._DI1.Done AND 
				FanucRobot._DI12.RSR1_Active 
			THEN
				uiShippingHomingStep := 1200;
			END_IF
			
	1200:	// 檢查手臂夾具的開合狀態
			TON_RobotRSR01_Delay.IN := FALSE;
			IF NOT fanucRobot._DI1.ClampA_Open THEN
				uiShippingHomingStep := 2000;
			ELSE
				uiShippingHomingStep := 9000;
			END_IF
			
	2000:	// 同尺寸軌道 busy Check
			TON_RobotFeedOutCommand.IN := TRUE;
			_fbShippingRobot_TransmitCVEnd.M_StartHomingFeedOut(UseA := TRUE);
			IF _fbShippingRobot_TransmitCVEnd.Busy THEN
				uiShippingHomingStep := 2100;
			END_IF
			IF TON_RobotFeedOutCommand.Q THEN
				iErrorID := 10;
			END_IF
	
	2100:	// 同尺寸軌道 done Check
			TON_RobotFeedOutCommand.IN := FALSE;
			TON_RobotTimeOut.IN := TRUE;
			IF _fbShippingRobot_TransmitCVEnd.Done THEN
				_fbShippingRobot_TransmitCVEnd.M_ResetHomingFeedOut();		
				uiShippingHomingStep := 0;
			END_IF
			IF TON_RobotTimeOut.Q THEN
				iErrorID := 11;
			END_IF

	9000:	// process done
			FanucRobotCheckTon.IN := FALSE;
			Homed := TRUE;
			xComplete := TRUE;
END_CASE

IF FanucRobotCheckTon.Q THEN
	iErrorID := 4;
END_IF
END_METHOD

METHOD ExitAction
VAR_INPUT
    xAfterCleanup : BOOL;
    xInCopyCode : BOOL;
END_VAR
END_METHOD

METHOD M_GetErrorMsg : T_MaxString
VAR_INPUT
	xErrorID: INT;
END_VAR

VAR
	
END_VAR
CASE xErrorID OF
    0:
        M_GetErrorMsg := 'No Error';
    1:
        M_GetErrorMsg := 'FB_ShippingHoming ErrorID 1: Action time out';
    2:
        M_GetErrorMsg := 'FB_ShippingHoming ErrorID 2: Cylinder not ready';
    3:
        M_GetErrorMsg := 'FB_ShippingHoming ErrorID 3: Motor not ready';
    4:
		M_GetErrorMsg := 'FB_ShippingHoming ErrorID 4: FanucRobot can not homing';
	10:
		M_GetErrorMsg := 'FB_ShippingHoming ErrorID 10: Shipping FanucRobot FeedOut to SameSizeConveyor not busy';
	11:
		M_GetErrorMsg := 'FB_ShippingHoming ErrorID 11: Shipping FanucRobot FeedOut to SameSizeConveyor Done Timeout';
	20:
		M_GetErrorMsg := 'FB_ShippingHoming ErrorID 20: Occupid , AutoMode_ShippingRobot_TransmitCVEnd in Executing ';
	21:
		M_GetErrorMsg := 'FB_ShippingHoming ErrorID 21: RSR02 Complete but FanucRobot still in Error';
	30:
		M_GetErrorMsg := 'FB_ShippingHoming ErrorID 30: Reboot ShippingArea FanucRobot Connect TimeOut';

END_CASE
END_METHOD

METHOD ResetAction
VAR_OUTPUT
    xComplete : BOOL := TRUE;
END_VAR
FanucRobotCheckTon.IN := FALSE;
TON_RobotRSR01_Delay.IN	:= FALSE;
TON_RebootPowerDelay.IN := FALSE;
TON_ConnectionTimeout.IN := FALSE;
TON_StartupDelay.IN		:= FALSE;
_fbShippingRobot_TransmitCVEnd.M_ResetHomingFeedOut();
END_METHOD

METHOD StartAction
VAR_OUTPUT
    xComplete : BOOL := TRUE;
	iErrorID : INT := 0;
END_VAR
Homed := FALSE;
FanucRobotCheckTon.IN 		:= FALSE;
ResetRobotDelay.IN 			:= FALSE;
TON_RobotFeedOutCommand.IN 	:= FALSE;
TON_RobotTimeOut.IN 		:= FALSE;
TON_RobotRSR01_Delay.IN		:= FALSE;
TON_RebootPowerDelay.IN		:= FALSE;
TON_ConnectionTimeout.IN	:= FALSE;
TON_StartupDelay.IN			:= FALSE;
uiShippingHomingStep := 0;
_fbShippingRobot_TransmitCVEnd.M_ResetHomingFeedOut();

IF  Service.AutoMode_ShippingRobot_TransmitCVEnd.Command.Execute AND
	Service.AutoMode_ShippingRobot_TransmitCVEnd.Status.Busy AND
	Service.AutoMode_ShippingRobot_TransmitCVEnd.Status.Error 
THEN
	iErrorID := 20;
END_IF
END_METHOD

END_FUNCTION_BLOCK

// ---- Library/20_MachineUnits/23_ShippingArea/RobotService/FB_ShippingRobot_TransmitCVEnd.TcPOU
FUNCTION_BLOCK FB_ShippingRobot_TransmitCVEnd EXTENDS FB_RobotRegionMove_BufferArea
VAR_INPUT
	INPUT       : REFERENCE TO ST_InputTable;
	Motor    	: REFERENCE TO UNI_MotorList;
	bCompleteRequest	: BOOL;
	fbSHippingHomingBusy	: BOOL;
END_VAR
VAR_OUTPUT
END_VAR
VAR
	//Area : E_RobotArea := E_RobotArea.TransmitCV_End;
	SensorToBeCheck :BIT;
	ConveyorMotor	: REFERENCE TO FB_Motor ;
	tonBoxArriveDelay 	: TON;
	BuzzBlink	:BLINK;
	LightBlink	:BLINK;
END_VAR

SUPER^.A10_StateControl();
A00_BasicUnits();
Area := E_RobotArea.TransmitCV_End;

ACTION A00_BasicUnits:
tonTimeOut(PT:=T#90S);
tonBoxArriveDelay(PT:=T#1S);

ErrorID:=2250;
END_ACTION

METHOD M_CheckCommand : BOOL // True : Command is useful
VAR_INPUT
END_VAR
VAR
	
END_VAR
// Check command paremeter is correct

IF fbShippingHomingBusy THEN
	THIS^.Get := info.Get;		//check Shipping Homing use
ELSE
	THIS^.Get :=TRUE; // For this service , robot only pick box from conveyor
END_IF

UseA := TRUE; // Only clip A avaliable
UseB := FALSE; // No clipB 	
		
	
	
CASE 	LREAL_TO_INT(Info.A_Position) OF	
	
1: // Pick box from Samesize conveyor
	SensorToBeCheck :=INPUT.bSameSizeCV_BoxNearShippingSensor;
	ConveyorMotor	REF= Motor.List.TransmitSameSideCV;
2: // Pick box from diffSize conveyor
	SensorToBeCheck :=INPUT.bDifferentSizeCV_BoxNearShippingSensor;
	ConveyorMotor	REF= Motor.List.TransmitDifferentSideCV;
ELSE
	strStatus:='FB_ShippingRobot_TransmitCVEnd: Wrong command ,Position A Not allow';
			M_CheckCommand:=FALSE;
			RETURN;	
END_CASE
		

IF Get THEN
	IF NOT Robot._DI1.ClampA_Open THEN
		strStatus := 'FB_ShippingRobot_TransmitCVEnd: Get command , clamp have box ';
		M_CheckCommand := FALSE;
		RETURN;
	END_IF
ELSE
	IF Robot._DI1.ClampA_Open THEN 
		strStatus := 'FB_ShippingRobot_TransmitCVEnd: Place command , clamp not have box ';
		M_CheckCommand := FALSE;
		RETURN;
	END_IF
END_IF


M_CheckCommand:=TRUE;
END_METHOD

METHOD M_CheckUnitsNotBusy : BOOL
VAR_INPUT
END_VAR
M_CheckUnitsNotBusy := true;
END_METHOD

METHOD M_CheckUnitsReady : BOOL
VAR_INPUT
END_VAR
M_CheckUnitsReady := true;
END_METHOD

METHOD M_ResetHomingFeedOut : BOOL
VAR_INPUT
END_VAR
Execute := FALSE;
info.UseA := FALSE;
info.UseB := FALSE;

M_ResetHomingFeedOut := TRUE;
END_METHOD

METHOD PRIVATE M_SensorUpdate : BOOL
VAR_INPUT
END_VAR
CASE 	LREAL_TO_INT(Info.A_Position) OF	
	
1: // Pick box from Samesize conveyor
	SensorToBeCheck :=INPUT.bSameSizeCV_BoxNearShippingSensor;
	
2: // Pick box from diffSize conveyor
	SensorToBeCheck :=INPUT.bDifferentSizeCV_BoxNearShippingSensor;

	
	END_CASE
END_METHOD

METHOD M_StartHomingFeedOut : BOOL
VAR_INPUT
	UseA	: BOOL;
END_VAR
// Place SameSize conveyor homing only place
Info.Get := FALSE;

Info.UseA 		:= UseA;
info.A_Position := 1;

Execute := TRUE;

M_StartHomingFeedOut := TRUE;
END_METHOD

METHOD  M_STATE_ABORTED
VAR_INPUT
END_VAR
ERROR :=TRUE;
Busy    := FALSE;
Aborted := TRUE;
Status := strStatus;
uiAbortingStep := 0;
_AbortCompleted := FALSE;
UniqueErrorCode:=_UniqueErrorCode;


IF NOT Execute THEN
	eSTATE:=STATE_RESETTING;
END_IF

IF Execute AND Reset THEN
	Error := FALSE;
	Aborted := false;
	uiExecutingStep :=uiResumeStep;
//	PreviousStrStatus := strStatus;
//	PreviousErrorCode := _UniqueErrorCode;
	Status := 'FB_ShippingRobot_TransmitCVEnd: no error';
	eSTATE:=STATE_EXECUTING;
END_IF
END_METHOD

METHOD  M_STATE_ABORTING
VAR_INPUT
END_VAR
CASE uiAbortingStep OF
	0 :
			_Abort 			:= FALSE;
			Abort 			:= FALSE;
			tonTimeOut.IN 	:= FALSE;
			uiAbortingStep	:= 9999;

			ConveyorMotor.M_MotorStop();
			
			
			
//			IF strStatus = PreviousStrStatus THEN
//				_UniqueErrorCode :=PreviousErrorCode;
//			END_IF
	9999:	
			_AbortCompleted:=TRUE;
END_CASE

IF _AbortCompleted THEN	
	eSTATE :=STATE_ABORTED;
END_IF
END_METHOD

METHOD  M_STATE_DONE
VAR_INPUT
END_VAR
Busy   := FALSE;
_Error := Error := FALSE;
_Abort := Abort := FALSE;
Done   := TRUE;

IF NOT Execute THEN
    eState := STATE_RESETTING;
END_IF
END_METHOD

METHOD  M_STATE_DORMANT
VAR_INPUT
END_VAR
// Clear FB output
Busy            := FALSE;
Done            := FALSE;
Aborted         := FALSE;
Error           := FALSE;
ErrorID         := 0;
Status          := '';
_ResetCompleted := FALSE;
_Error          := FALSE;
_Executed       := FALSE;

tonTimeOut.IN:=FALSE;
tonBoxArriveDelay.IN :=FALSE;
strStatus :='FB_ShippingRobot_TransmitCVEnd: No Error';
uiExecutingStep :=uiResettingStep :=uiResumeStep :=0;
PreviousStrStatus			 :='';
PreviousErrorCode			 :='';
_UniqueErrorCode	:='0';

// Wait Execute command
IF Execute THEN
    eState := STATE_EXECUTING;
END_IF
END_METHOD

METHOD  M_STATE_ERROR
VAR_INPUT
END_VAR
ERROR   :=TRUE;
Busy	:=FALSE;
Status := strStatus;
UniqueErrorCode:=_UniqueErrorCode;
IF info.A_Position = 1 OR 
	info.A_Position = 2 THEN
	ConveyorMotor.M_MotorStop();
END_IF

IF NOT Execute THEN	
eSTATE:=STATE_RESETTING;
END_IF
END_METHOD

METHOD  M_STATE_EXECUTING
VAR_INPUT
END_VAR
VAR_INST
    ActionMode       : E_ReloadRoundBoxAction;
	BoxReady_1st : BOOL;
	BoxReady_2nd : BOOL;
    CarrierReady_1st : BOOL;
    CarrierReady_2nd : BOOL;
    uiBothStep : UINT;
    uiSingleClampStep : UINT;
	Address_A : INT;
	Address_B : INT;
	bMoveConveyorForward	: BOOL;
	bMoveConveyorBackward	: BOOL;
	
END_VAR
VAR
	WareHouse: INT;
END_VAR
// Set Busy active edit by johnson
Busy := TRUE;
M_SensorUpdate();

IF THIS^.Stop THEN // Pending the timeout when Stop signal occur
	tonTimeout.IN :=FALSE;
END_IF

IF bMoveConveyorForward THEN
	IF NOT ConveyorMotor.InBackWard THEN
		ConveyorMotor.M_MoveForward();
	END_IF
END_IF

IF bMoveConveyorBackward THEN
	IF NOT ConveyorMotor.InForWard THEN
		ConveyorMotor.M_MoveBackward();
	END_IF
	
END_IF
// Service Process
CASE uiExecutingStep OF
	0:
			// Clear variable
			bMoveConveyorForward := FALSE;
			ActionMode       := E_ReloadRoundBoxAction.Undefined;
			CarrierReady_1st := FALSE;
			CarrierReady_2nd := FALSE;
			uiBothStep := 0;
			uiSingleClampStep :=0;
			BoxReady_1st := 0;
			BoxReady_2nd := 0;
			tonTimeOut.IN:=FALSE;
			// Check command
			IF M_CheckCommand() THEN
				uiExecutingStep := 10;
			ELSE
				_Error:=TRUE;
			END_IF
    10:
			// Start process, check units first
			IF M_CheckUnitsReady() THEN
				uiExecutingStep := 20;
			END_IF
    20:
			// CHeck units not busy state
			IF M_CheckUnitsNotBusy() THEN
				uiExecutingStep := 50;
			END_IF
	50:
			IF Get THEN
				uiExecutingStep := 100;
			ELSIF NOT Get  THEN
				uiExecutingStep := 500;
			ELSE
				strStatus := 'FB_ShippingRobot_TransmitCVEnd Step 50: Wrong command';
				_Error 	  := TRUE;
			END_IF
   
	100: //Move conveyor 
			bMoveConveyorForward:=TRUE;
			ConveyorMotor.M_MoveForward();			
			uiExecutingStep := 1000;	

	500:
			bMoveConveyorBackward := TRUE;
			IF ConveyorMotor.InBackWard AND NOT SensorToBeCheck THEN
				uiExecutingStep := 1000;
			END_IF
	
	1000:   
			// Read   coordinate
 			 Address_A := LREAL_TO_INT(Info.A_Position);
			 Address_B := LREAL_TO_INT(Info.B_Position);
			 
			IF UseA AND NOT UseB THEN
				//Only clampA
				uiExecutingStep := 10000;
			END_IF
       
    10000: // Only ClampA 
			IF NOT Robot._DI1.Done THEN            
					IF Get THEN
						tonBoxArriveDelay.IN := SensorToBeCheck;      	
					ELSIF fbSHippingHomingBusy AND NOT Get THEN
						BoxReady_1st:=TRUE;				// Only ShippingHoming FeedOut Use
					END_IF	 
					  // Robot Abs move
					 Robot.M_StartRobotAbsMove(GetBox:=Get,
												UseClampA:=UseA,
												UseClampB:=UseB,
												Area:=Area,
												ClampA_Address:=Address_A,
												ClampB_Address:=Address_B,
												BoxReady_1:=tonBoxArriveDelay.Q OR BoxReady_1st,
												BoxReady_2:=BoxReady_2nd);	  
			
			ELSE
				tonTimeOut.IN:=FALSE;
				tonBoxArriveDelay.IN :=FALSE;
				uiExecutingStep := 10080;
			END_IF
				tonTimeOut.IN:=TRUE;
				IF tonTimeOut.Q=TRUE THEN		
					uiResumeStep  	:= 10000;	
					strStatus 		:='FB_ShippingRobot_TransmitCVEnd Step 10000: wait Box Arrived TransCV time out';
					_Abort			:= TRUE;
				END_IF	
    10080:
			Robot.M_ResetRobotAbsMove(UseA,UseB); // Clear command and go to place box
			tonTimeOut.IN:=TRUE;
			IF NOT Robot._DI1.Done THEN
				tonTimeOut.IN:=FALSE;
				uiExecutingStep := 90000; 
			END_IF
			IF tonTimeOut.Q=TRUE THEN
				uiExecutingStep := 10080;
				strStatus 		:='FB_ShippingRobot_TransmitCVEnd Step 10080: Reset Robot timeout';
				_Abort			:= TRUE;
			END_IF	
    
   90000:
			bMoveConveyorForward  := FALSE;
			bMoveConveyorBackward := FALSE;
			ConveyorMotor.M_MotorStop();
			IF ConveyorMotor.InStopped THEN
				uiExecutingStep := 99000;
			END_IF
		
    99000: // process done
                Status    := 'FB_ShippingRobot_TransmitCVEnd Step 99000: Process completed';
        		_Executed := TRUE;
END_CASE

// State Control
IF _Executed THEN
    eState := STATE_DONE;
ELSIF _Error THEN
    eState := STATE_ERROR;
ELSIF NOT Execute THEN
    eState := STATE_RESETTING;
END_IF
IF _Abort OR Abort THEN
	eSTATE:=STATE_ABORTING;
END_IF
END_METHOD

METHOD  M_STATE_RESETTING
VAR_INPUT
END_VAR
// Done := false 更改到Dormant 清除確保，上位檢查到done 後可以直接下Execute


CASE uiResettingStep OF

	0:
		tonTimeOut.IN:=FALSE;
		ConveyorMotor.M_MotorStop();

//		Robot.M_ResetRobotAbsMove(TRUE,TRUE);

		uiResettingStep:=100;

	100:
		Robot.M_ResetAllCommand();
		IF Robot.M_CheckResetAllCommand() THEN
			uiResettingStep := 9999;
		END_IF

	9999:
		_ResetCompleted:=TRUE;
END_CASE
IF _ResetCompleted THEN
	eSTATE:=STATE_DORMANT;
END_IF
END_METHOD

END_FUNCTION_BLOCK

// ---- Library/20_MachineUnits/23_ShippingArea/RobotService/FB_ShippingRobot_Left.TcPOU
FUNCTION_BLOCK FB_ShippingRobot_Left EXTENDS FB_RobotRegionMove_BufferArea
VAR_INPUT
	Buzz	: REFERENCE TO BOOL;
	RedLamp	: REFERENCE TO BOOL;
	bCompleteRequest	: BOOL;
	Input		: REFERENCE TO ST_InputTable;
END_VAR
VAR_OUTPUT
	bTransCVInPosition	: BOOL;
END_VAR
VAR
	//Area : E_RobotArea := E_RobotArea.TransmitCV_End;
	Blink		: ST_BlinkInfo;
	BuzzBlinker	: Blink;
	LightBlinker: Blink;
	TrigBuzz	: R_TRIG;
	TrigLight	: R_TRIG;
	BlinkInfo	: ST_BlinkInfo;
	
	TON_BlinkDelay	: TON;
END_VAR

SUPER^.A10_StateControl();
A00_BasicUnits();
Area := E_RobotArea.ShippingRobotLeft;

ACTION A00_BasicUnits:
tonTimeOut(PT:=T#60S);
TON_BlinkDelay(PT:=T#1S);

bTransCVInPosition := Input.bShippingTransCV_Leftside_Arrived;
ErrorID:=2250;
END_ACTION

METHOD M_CheckCommand : BOOL // True : Command is useful
VAR_INPUT
END_VAR
VAR
	
END_VAR
// Check command paremeter is correct

THIS^.Get :=Info.Get;
UseA := Info.UseA;
UseB := Info.UseB;
//Buffer area
		
IF UseA AND ( Info.A_Position<1 OR  Info.A_Position>40) THEN
	strStatus:='FB_ShippingRobot_Left: Wrong command ,Position A Not allow';
	M_CheckCommand:=FALSE;
	RETURN;			
END_IF		

IF UseB AND( Info.B_Position<1 OR  Info.B_Position>40 )THEN
	strStatus:='FB_ShippingRobot_Left: Wrong command ,Position B Not allow';
	M_CheckCommand:=FALSE;
	RETURN;			
END_IF

IF Get THEN
	IF NOT Robot._DI1.ClampA_Open THEN
		strStatus := 'FB_ShippingRobot_Left: Get command , clamp have box ';
		M_CheckCommand := FALSE;
		RETURN;
	END_IF
ELSE
	IF Robot._DI1.ClampA_Open THEN 
		strStatus := 'FB_ShippingRobot_Left: Place command , clamp not have box ';
		M_CheckCommand := FALSE;
		RETURN;
	END_IF
END_IF
		
M_CheckCommand:=TRUE;
END_METHOD

METHOD M_CheckUnitsNotBusy : BOOL
VAR_INPUT
END_VAR
M_CheckUnitsNotBusy := true;
END_METHOD

METHOD M_CheckUnitsReady : BOOL
VAR_INPUT
END_VAR
M_CheckUnitsReady := true;
END_METHOD

METHOD  M_STATE_ABORTED
VAR_INPUT
END_VAR
ERROR :=TRUE;
Busy    := FALSE;
Aborted := TRUE;
Status := strStatus;
_AbortCompleted := FALSE;
uiAbortingStep := 0;
UniqueErrorCode:=_UniqueErrorCode;
IF NOT Execute THEN
	eSTATE:=STATE_RESETTING;
END_IF

IF Execute AND Reset THEN
		Error := FALSE;
	Aborted := false;
	uiExecutingStep :=uiResumeStep;
	PreviousStrStatus := strStatus;
	PreviousErrorCode := _UniqueErrorCode;
	eSTATE:=STATE_EXECUTING;
END_IF
END_METHOD

METHOD  M_STATE_ABORTING
VAR_INPUT
END_VAR
CASE uiAbortingStep OF
	0 :
		tonTimeOut.IN 	:= FALSE;
		Abort 			:= false;
		_Abort 			:= FALSE;
		uiAbortingStep:=9999;
		
		IF strStatus = PreviousStrStatus THEN
			_UniqueErrorCode :=PreviousErrorCode;
		END_IF
		
	9999:	_AbortCompleted:=TRUE;
END_CASE

IF _AbortCompleted THEN	
	eSTATE :=STATE_ABORTED;
END_IF
END_METHOD

METHOD  M_STATE_DONE
VAR_INPUT
END_VAR
Busy   := FALSE;
_Error := Error := FALSE;
_Abort := Abort := FALSE;
Done   := TRUE;

IF NOT Execute THEN
    eState := STATE_RESETTING;
END_IF
END_METHOD

METHOD  M_STATE_DORMANT
VAR_INPUT
END_VAR
// Clear FB output
Busy            := FALSE;
Done            := FALSE;
Aborted         := FALSE;
Error           := FALSE;
ErrorID         := 0;
Status          := '';
_ResetCompleted := FALSE;
_Error          := FALSE;
_Executed       := FALSE;

bCompleteRequest := false;
tonTimeOut.IN:=FALSE;
TON_BlinkDelay.IN := FALSE;
strStatus :='No Error';
uiExecutingStep :=uiResettingStep :=uiResumeStep :=0;
PreviousStrStatus			 :='';
PreviousErrorCode			 :='';
_UniqueErrorCode	:='0';

// Wait Execute command
IF Execute AND bTransCVInPosition THEN
    eState := STATE_EXECUTING;
ELSE
	strStatus :='FB_ShippingRobot_Left: Wrong command ,TransCV not In Position ';
	_Error:= TRUE;
END_IF
END_METHOD

METHOD  M_STATE_ERROR
VAR_INPUT
END_VAR
ERROR   :=TRUE;
Busy	:=FALSE;
Status := strStatus;
UniqueErrorCode:=_UniqueErrorCode;
IF NOT Execute THEN	
eSTATE:=STATE_RESETTING;
END_IF
END_METHOD

METHOD  M_STATE_EXECUTING
VAR_INPUT
END_VAR
VAR_INST
    ActionMode       : E_ReloadRoundBoxAction;
	BoxReady_1st : BOOL;
	BoxReady_2nd : BOOL;
    CarrierReady_1st : BOOL;
    CarrierReady_2nd : BOOL;
    uiBothStep : UINT;
    uiSingleClampStep : UINT;
	Address_A : INT;
	Address_B : INT;
	
END_VAR
VAR
	WareHouse: INT;
END_VAR
// Set Busy active edit by johnson
Busy := TRUE;
IF THIS^.Stop THEN // Pending the timeout when Stop signal occur
	tonTimeout.IN :=FALSE;
END_IF
// Service Process
CASE uiExecutingStep OF
	0:
        // Clear variable
        ActionMode       := E_ReloadRoundBoxAction.Undefined;
        CarrierReady_1st := FALSE;
        CarrierReady_2nd := FALSE;
        uiBothStep := 0;
		uiSingleClampStep :=0;
		BoxReady_1st := 0;
		BoxReady_2nd := 0;
		tonTimeOut.IN:=FALSE;
        // Check command
        IF M_CheckCommand() THEN
            uiExecutingStep := 10;
		ELSE
			_Error:=TRUE;
        END_IF
    10:
        // Start process, check units first
        IF M_CheckUnitsReady() THEN
            uiExecutingStep := 20;
        END_IF
    20:
        // CHeck units not busy state
        IF M_CheckUnitsNotBusy() THEN
            uiExecutingStep := 1000;
        END_IF
   
	1000:   
			// Read   coordinate
 			 Address_A := LREAL_TO_INT(Info.A_Position);
			 Address_B := LREAL_TO_INT(Info.B_Position);
			 
			IF UseA AND NOT UseB THEN
				//Only clampA
				uiExecutingStep := 10000;
			ELSIF NOT UseA AND UseB THEN
				//Only ClampB 
				uiExecutingStep := 20000;
			ELSIF UseA AND UseB THEN
				//Both Clamps
				uiExecutingStep := 30000;		
			END_IF
       
    10000: // Only ClampA 
        IF NOT Robot._DI1.Done THEN            
           		BoxReady_1st:=TRUE;				
			          		 
				  // Robot Abs move
           		 Robot.M_StartRobotAbsMove(GetBox:=Get,
											UseClampA:=UseA,
											UseClampB:=UseB,
											Area:=Area,
											ClampA_Address:=Address_A,
											ClampB_Address:=Address_B,
											BoxReady_1:=BoxReady_1st,
											BoxReady_2:=BoxReady_2nd);	  
		
        ELSE
			tonTimeOut.IN:=FALSE;
            uiExecutingStep := 10080;
        END_IF
		
		tonTimeOut.IN:=TRUE;
		IF tonTimeOut.Q THEN
			tonTimeOut.IN:=FALSE;
			uiResettingStep := 10000;
			strStatus :='FB_ShippingRobot_Left Step 10000: Reset Robot timeout';
			_Abort:=TRUE;
		END_IF
		IF Robot.Error THEN
			uiResettingStep := 10000;
			strStatus := CONCAT('FB_ShippingRobot place Left Plate Error',robot.ErrMsg);
			_Abort := TRUE;
		END_IF
    10080:
        Robot.M_ResetRobotAbsMove(UseA,UseB); // Clear command and go to place box
		tonTimeOut.IN:=TRUE;
        IF NOT Robot._DI1.Done THEN
			tonTimeOut.IN:=FALSE;
            uiExecutingStep := 90000; 
        END_IF
    	IF tonTimeOut.Q=TRUE THEN
			uiResettingStep := 10080;
			strStatus :='FB_ShippingRobot_Left Step 10080: Reset Robot timeout';
			_Abort:=TRUE;
		END_IF

   20000: // Only ClampB
        IF NOT Robot._DI1.Done THEN           		
				BoxReady_2nd:=TRUE;				          		 
				  // Robot Abs move
           		 Robot.M_StartRobotAbsMove( GetBox:=Get,
											UseClampA:=UseA,
											UseClampB:=UseB,
											Area:=Area,
											ClampA_Address:=Address_A,
											ClampB_Address:=Address_B,
											BoxReady_1:=BoxReady_1st,
											BoxReady_2:=BoxReady_2nd);	
        ELSE
			tonTimeOut.IN:=FALSE;
            uiExecutingStep := 20080;
        END_IF
		tonTimeOut.IN:=TRUE;
			IF tonTimeOut.Q=TRUE THEN
				tonTimeOut.IN:=FALSE;
				strStatus :='FB_ShippingRobot_Left Step 20000: Reset Robot timeout';
				_Error:=TRUE;
			END_IF
    20080:
       Robot.M_ResetRobotAbsMove(UseA,UseB);; // Clear command 

        IF NOT Robot._DI1.Done THEN
            uiExecutingStep := 90000; 
        END_IF
		tonTimeOut.IN:=TRUE;
		IF tonTimeOut.Q=TRUE THEN
			strStatus :='FB_ShippingRobot_Left Step 20080: Reset Robot timeout';
			_Error:=TRUE;
		END_IF
    30000: // Both Clamps
        		
		
